// Transfermode/specific_MA_config/FB_Write_config_MA_06
/// This function block can be used to download the configuration of Motion App 6 ("ECO drive").
/// The specific parameters of this Motion App are the inputs of this FB and can be defined by the user. 
/// The function block uses the transfer mode to write this configuration to the Motion Terminal
/// and indicates the state of the download process.

FUNCTION_BLOCK FB_Write_config_MA_06
VAR_INPUT
	awBusDataFromVTEM 				: ARRAY [0..2] OF WORD;		(* 6 bytes of process data received from the Motion Terminal *)
END_VAR
	
VAR_IN_OUT
	awBusDataToVTEM 				: ARRAY [0..2] OF WORD; 	(* 6 bytes of process data sent to the Motion Terminal *)
END_VAR

VAR_INPUT
	xExecute 						: BOOL; 					(* has to be set to TRUE for a download and to FALSE to reset the function block after a download *)

	iParameterSet					: INT := 1; 				(* the parameter set to be written to, 1 by default *)
	
	// system parameters
		iInPortRetracted			: INT;						// Sensor port for detection of end position at pressurisation of outlet port 2 (retracted), value is number of the slot (beginning from 0 and including valve slots) * 10 + number of the port
		iInPortAdvanced				: INT;						// Sensor port for detection of end position at pressurisation of outlet port 4 (advanced), value is number of the slot (beginning from 0 and including valve slots) * 10 + number of the port

END_VAR

VAR_OUTPUT                  		
	iResponse 						: eTransferResponse; 		(* returns the status of the execution of the download process *)
	sCurrentValue 					: STRING; 					(* indicates which value of the array is currently treated (necessary to evaluate in case of error messages) *)
	xDownloadDone 					: BOOL; 					(* indicates whether the download was successful *)
	xDownloadError 					: BOOL := FALSE; 			(* indicates whether an error occurred during the transfer *)
END_VAR

VAR
	aTransferPackages				: ARRAY [0..100] OF stTransferPackage;
	fbdownloadMultipleParameters 	: FB_Download_Multiple_Parameters;
	iCurrentValue					: INT;
	fbWriteValueToWord 				: FB_Write_Value_To_Word;
END_VAR

(*****************************************************************************************************

Festo SE & Co. KG, Esslingen
Copyright (c) 2018. All rights reserved.

Product:            Motion Terminal VTEM
Description:        Function Block to download the parameters for Motion App 6 to the Motion Terminal

Object version:     2.00
Last change:        2019-03
======================================================================================================
                                       H I S T O R Y
======================================================================================================
Version:            2.00
Date:               2019-03
Change/Activity:    - created (#2368895)
Release:            3.5.7.230 (CODESYS 3.5.7.2, Lib version 3.0)
Author:             JEBU
======================================================================================================

*****************************************************************************************************)

// write the Motion App specific parameters into the struct
	//iInPortRetract
		aTransferPackages[0].iChannel := iParameterSet;
		aTransferPackages[0].iAddressedTarget := 6;
		aTransferPackages[0].iIndex := 70;
		aTransferPackages[0].iTransferValue := iInPortRetracted;
	
	//iInPortRetract
		aTransferPackages[1].iChannel := iParameterSet;
		aTransferPackages[1].iAddressedTarget := 6;
		aTransferPackages[1].iIndex := 71;
		aTransferPackages[1].iTransferValue := iInPortAdvanced;
	
	// define end of parameter list to be downloaded by setting all variables to 0 (end criterion for FB_Download_Multiple_Parameters)
		aTransferPackages[2].iChannel := 0;
		aTransferPackages[2].iAddressedTarget := 0;
		aTransferPackages[2].iIndex := 0;
		aTransferPackages[2].iTransferValue := 0;


// pre-check of the value for the parameter set
	IF xExecute = TRUE AND (iParameterSet < 1 OR iParameterSet > 5) THEN		// invalid input for the parameter set
		xDownloadDone := FALSE; 
		xDownloadError := TRUE; 
		iResponse := eTransferResponse.invalid_ParameterSet; 
		iCurrentValue := 0; 
		// send command 'stop'
		fbWriteValueToWord(iValue := 61, iStartBit := 0, iEndBit := 5, wDataWord := awBusDataToVTEM[0]); 			// ValveMode = 61
		fbWriteValueToWord(iValue := 0, iStartBit := 6, iEndBit := 15, wDataWord := awBusDataToVTEM[0]); 			// (empty)
		awBusDataToVTEM[1] := 0; 
		awBusDataToVTEM[2] := 0; 
		
	ELSE	
		// call the function block for multiple parameter download
			fbdownloadMultipleParameters(	xExecute := xExecute,
											awBusDataFromVTEM := awBusDataFromVTEM,
											aTransferPackages := aTransferPackages, 
											awBusDataToVTEM := awBusDataToVTEM,
											xDownloadDone => xDownloadDone,
											xDownloadError => xDownloadError,
											iResponse => iResponse,
											iCurrentValue => iCurrentValue);
	END_IF
	
	
// The current value output is needed if there is any invalid value in order to address it correctly.
// As the user doesn't work with indices in this function block, the current value is transformed to a string holding the name of the parameter.
	CASE iCurrentValue OF
		0: sCurrentValue := 'iInPortRetract';
		1: sCurrentValue := 'iInPortAdvanced';
		2: sCurrentValue := 'AllParametersWritten';
	END_CASE

END_FUNCTION_BLOCK

// Operation/FB_TeachInRun
/// This function block is designed to execute the teach-in run (Valve Mode 60) on a valve. 
/// Before executing the transfer mode, the Parameter 255 (Motion App to be tought in) is
/// parameterised with the value on the corresponding input.
/// After that the teach-in run is started and can be controlled via the input "iManualControl"
/// if the manual operation is possible for the selectes Motion App.

FUNCTION_BLOCK FB_TeachInRun
VAR_INPUT
	awBusDataFromVTEM				: ARRAY [0..2] OF WORD;				// 6 bytes of process data that is received from the Motion Terminal
END_VAR

VAR_IN_OUT
	awBusDataToVTEM					: ARRAY [0..2] OF WORD;				// 6 bytes of process data that is sent to the Motion Terminal
END_VAR

VAR_INPUT
	xEnable							: BOOL;								// has to be set to TRUE in order to operate the teach-in run on the valve, otherwise the teach-in run is stopped  
	iParameterSet					: INT;								// Parameter Set to be used for storing the learning data (0 = current parameter set, 1…5 = parameter set 1…5)
	iMotionAppToBeToughtIn			: INT;								// ID of the Motion App that is to be taught-in
	iOperatingMode					: INT;								// Sets operating mode of teach-in run (0 = Stop, 1 = Auto, 2 = Manual (only Motion App #11)
	iManualControl					: INT;								// Control input for manual execution of teach-in run (0 = Block, 1 = Advance, 2 = Retract, 3 = Exhaust)
	xAcknowledge					: BOOL;								// errors can be acknowledged (after they got inactive) with a rising edge at this input, while the FB is enabled
END_VAR

VAR_OUTPUT
	xDone							: BOOL;								// indicates that the teach-in run was finished successfully
	xError							: BOOL;								// indicates that an Error occured
	iResponse						: eResponseTeachInRun;				// returns the status of the TeachInRun function block
	sResponseDescription			: STRING;							// returns the status of the TeachInRun function block as string
	xWarning						: BOOL;								// indicates whether there is a warning returned by the teach-in run
	xRetractedEndPos_optional		: BOOL;								// only if digital sensors are installed (optional): indicates whether the retracted end position was reached (after outlet port 2 is pressurised)
	xAdvancedEndPos_optional		: BOOL;								// only if digital sensors are installed (optional): indicates whether the advanced end position was reached (after outlet port 4 is pressurised)
END_VAR

VAR
	// State machine variables
		iState						: INT := 10;						// Value for the local state machine
		xStateChange				: BOOL;								// TRUE if the state is to be changed
		iCommandNumber				: INT;								// Value for the command case

	// First Cycle variables
		iParameterSetFC				: INT;								// Variable to store value from first cycle
		iMotionAppToBeToughtInFC	: INT;								// Variable to store value from first cycle
		iOperatingModeFCC			: INT;								// Variable to store value from first cycle in state "Completed" or "Error"
		iManualControlFCC			: INT;								// Variable to store value from first cycle in state "Completed" or "Error"

	// Function block instances
		fbreadbitsfromword				: FB_Read_Bits_From_Word;			// 
		fbwritevaluetoword				: FB_Write_Value_To_Word;			//
		fbstateinterpreterteachinrun	: FB_StateInterpreter_TeachInRun;	//

	// Current Valve variables
		iCurrentValveMode			: INT;									// 
		iCurrentValveState			: INT;									//
		iCurrentAppState			: INT;									//
		iCurrentChannelTM			: INT;									//
		iCurrentAddressedTargetTM	: INT;									//
		iCurrentIndexTM				: INT;									//
		iCurrentValueTM				: INT;									//
		iCurrentTransferControlTM	: INT;									//
		
	// Misc variables
		xInputValid					: BOOL;									// TRUE if the values iParameterSet, iMotionAppToBeToughtIn and iOperatingMode are within valid range
		xInputConsistent			: BOOL;
		xInvalidCommand				: BOOL;
		iInvalidCommand				: INT;
		xNoValve					: BOOL;
		xWebConfigAccess			: BOOL;
		xInvalidMotionApp			: BOOL;
		
		xAcknowledgeLastCycle		: BOOL;
		
		xAcknowledgeCompleted		: BOOL;
		xReadyToComplete			: BOOL;									// Indicator which shows that no outdated response of the last executed learning trip is evaluated. 
		xStateFinished				: BOOL;
		xStateError					: BOOL;
		
		iReadParameterSet			: INT;
		iWriteParameterSet			: INT;
		xReturnReadParameterSet		: BOOL;
		
		iCounter					: INT;
		iCounterMax					: INT := 3000;
		
		xTeachInRunWasActive		: BOOL;
END_VAR

(*****************************************************************************************************

Festo SE & Co. KG, Esslingen
Copyright (c) 2019. All rights reserved.

Product:            Motion Terminal VTEM
Description:        Function block to execute the teach-in run

Object version:     1.05
Last change:        2020-12
======================================================================================================
                                       H I S T O R Y
======================================================================================================
Version:            1.05 
Date:               2020-12        
Change/Activity:    - integrated new app state return values #10 and #11 (#3800494)
Release:            3.5.7.236
Author:             JEBU
------------------------------------------------------------------------------------------------------
Version:            1.04 
Date:               2020-05        
Change/Activity:    - created (#2256363)
Release:            3.5.7.234
Author:             JEBU/MKLP
======================================================================================================

******************************************************************************************************)

// Read the current status of the the motion terminal
	fbreadbitsfromword(wData:= awBusDataFromVTEM[0], iStartBit:=0, iEndBit:= 5, iValue=> iCurrentValveMode, xError=> );						// read current valve mode
	fbreadbitsfromword(wData:= awBusDataFromVTEM[0], iStartBit:=6, iEndBit:= 7, iValue=> iCurrentValveState, xError=> );					// read current valve state

	IF iCurrentValveMode <> 63 THEN																										// Operating mode:
		fbreadbitsfromword(wData:= awBusDataFromVTEM[0], iStartBit:=8, iEndBit:= 15, iValue=> iCurrentAppState, xError=>);					// read app state
	ELSIF iCurrentValveMode = 63 THEN																									// Transfer mode:
		fbreadbitsfromword(wData:= awBusDataFromVTEM[0], iStartBit:= 8, iEndBit:= 12, iValue=> iCurrentChannelTM, xError=> );				// read current channel
		fbreadbitsfromword(wData:= awBusDataFromVTEM[0], iStartBit:= 13, iEndBit:= 15, iValue=> iCurrentTransferControlTM, xError=> );		// read current transfer control
		fbreadbitsfromword(wData:= awBusDataFromVTEM[1], iStartBit:= 0, iEndBit:= 7, iValue=> iCurrentAddressedTargetTM, xError=> );		// read current addressed target
		fbreadbitsfromword(wData:= awBusDataFromVTEM[1], iStartBit:= 8, iEndBit:= 15, iValue=> iCurrentIndexTM, xError=> );					// read current index
		fbreadbitsfromword(wData:= awBusDataFromVTEM[2], iStartBit:= 0, iEndBit:= 15, iValue=> iCurrentValueTM, xError=> );					// read current value
	END_IF
	
	IF iCurrentValveMode = 60 AND iState = 40 THEN
		fbstateinterpreterteachinrun.byActualAppState := INT_TO_BYTE(iCurrentAppState);
		
		fbstateinterpreterteachinrun();
				
		xRetractedEndPos_optional := fbstateinterpreterteachinrun.xRetractedEndPos_optional;
		xAdvancedEndPos_optional := fbstateinterpreterteachinrun.xAdvancedEndPos_optional;
		xWarning := fbstateinterpreterteachinrun.xWarning;
		iResponse := fbstateinterpreterteachinrun.iTeachInRunState;
	END_IF
//-----------------------------------------------------------------------------------------------------------

// Transition for RESETTING 
	IF xEnable = FALSE AND iState <> 10 AND iState <> 100 THEN
		xStateChange := TRUE;
		iState := 100;
	END_IF
//-----------------------------------------------------------------------------------------------------------

// Transition for WebConfig Access denied
	IF 	xWebConfigAccess = FALSE AND 
		xEnable = TRUE AND iState <> 10 AND 
		iCurrentValveMode = 61 AND iCurrentAppState = 10 THEN 	// The WebConfig has write permission -> access denied for the PLC
			xStateChange := TRUE;
			iState := 70;
			xWebConfigAccess := TRUE;
	END_IF
//-----------------------------------------------------------------------------------------------------------
	
// Check if input data is consisent (not in state 10 IDLE)
	IF 	xInputConsistent = TRUE  AND 
		xEnable = TRUE AND iState <> 10 AND iState <> 15 AND 
		(iParameterSet <> iParameterSetFC OR iMotionAppToBeToughtIn <> iMotionAppToBeToughtInFC OR (iState = 70 AND xStateChange = FALSE AND (iOperatingModeFCC <> iOperatingMode OR iManualControlFCC <> iManualControl))) THEN
			xStateChange := TRUE;
			iState := 70;		// Input data inconsistent
			xInputConsistent := FALSE;		
	END_IF
	
	IF xNoValve = FALSE AND 
	   xEnable = TRUE AND iState <> 10 AND iState <> 15 AND 
	   iCurrentValveMode = 61 AND iCurrentValveState = 1 AND iCurrentAppState = 15 THEN		// no Valve detected 
			xNoValve := TRUE;
			xStateChange := TRUE;
			iState := 70;
	END_IF
//-----------------------------------------------------------------------------------------------------------

// Local state machine
	CASE iState OF
		10:	// IDLE mode
			// code that is executed only in the first cycle of this state
				IF xStateChange = TRUE THEN
					xStateChange := FALSE;
				END_IF
			//-----------------------------------------------------------------------------------------------------------
			
			// code that is repeated every cycle in this state	
				iCommandNumber := 0;	// IDLE
				iResponse := eResponseTeachInRun.idle;
			//-----------------------------------------------------------------------------------------------------------
			
			// Transition
				IF xEnable = TRUE THEN
					xStateChange := TRUE;	// Leave this state
					iState := 15;
				END_IF
			//-----------------------------------------------------------------------------------------------------------

		15:	// check validity and save values of "first cycle"
			// code that is executed only in the first cycle of this state
				IF xStateChange = TRUE THEN
					xStateChange := FALSE;
					iResponse := eResponseTeachInRun.storing_first_cycle_input_data;
					xInputConsistent := TRUE;
					iParameterSetFC := iParameterSet;
					iMotionAppToBeToughtInFC := iMotionAppToBeToughtIn;
				END_IF
			//-----------------------------------------------------------------------------------------------------------
			
			// code that is repeated every cycle in this state	
				IF (iParameterSet >= 0 AND iParameterSet <= 5) AND (iMotionAppToBeToughtIn >= 1 AND iMotionAppToBeToughtIn <= 59) AND (iOperatingMode >= 0 AND iOperatingMode <= 3) THEN
					xInputValid := TRUE;
				ELSE
					xInputValid := FALSE;
				END_IF
			//-----------------------------------------------------------------------------------------------------------
			
			// Transition
				IF xInputValid = TRUE THEN
					xStateChange := TRUE;	// Leave this state
					iState := 20;
				ELSE
					xStateChange := TRUE;	// Leave this state
					iState := 70;			// Failure
				END_IF
			//-----------------------------------------------------------------------------------------------------------
		
		20:	// Resetting valve mode to 61
			// code that is executed only in the first cycle of this state
				IF xStateChange = TRUE THEN
					xStateChange := FALSE;
					iResponse := eResponseTeachInRun.resetting_valve_to_61;
				END_IF
			//-----------------------------------------------------------------------------------------------------------
			
			// code that is repeated every cycle in this state	
				IF iCurrentValveMode = 63 THEN
					iCommandNumber := 1;	// exit transfer mode
				ELSIF iCurrentValveMode <> 61 AND iCurrentValveMode <> 63 AND iCurrentValveState = eValveState.Running THEN
					iCommandNumber := 2;	// stop running motion apps
				END_IF 
			//-----------------------------------------------------------------------------------------------------------
			
			// Transition
				IF iCurrentValveMode = 61 AND iCurrentValveState = eValveState.configurable THEN
					xStateChange := TRUE;	// Leave this state
					iState := 30;
				ELSIF iCurrentValveState = eValveState.NotReady OR iCurrentValveState = eValveState.Failure THEN
					xStateChange := TRUE;
					iState := 70;
				END_IF
			//-----------------------------------------------------------------------------------------------------------

		30: // Sending command to read active ParameterSet
				// code that is executed only in the first cycle of this state
				IF xStateChange = TRUE THEN
					xStateChange := FALSE;
					xStateFinished := FALSE;
					iResponse := eResponseTeachInRun.ReadingActiveParameterSet;
					iCommandNumber := 3;	// read active ParameterSet
				END_IF
			//-----------------------------------------------------------------------------------------------------------
			
			// code that is repeated every cycle in this state
				IF iCurrentValveMode = 63 AND iCurrentChannelTM = 15 AND iCurrentAddressedTargetTM = 0 AND iCurrentIndexTM = 1 THEN
					xStateFinished := TRUE;
					iReadParameterSet := iCurrentValueTM;
				ELSE // timeout mechanism after <iCounterMax> cycles within this state
					iCounter := iCounter + 1;
					IF iCounter = iCounterMax THEN
						xStateError := TRUE;
					END_IF
				END_IF
				
				IF iParameterSet = 0 THEN
					iWriteParameterSet := iReadParameterSet;
				ELSE
					iWriteParameterSet := iParameterSet;
				END_IF
			//-----------------------------------------------------------------------------------------------------------
				
			// Transition
				IF xStateFinished = TRUE THEN
					xStateChange := TRUE;
					iState := 32;
				ELSIF xStateError = TRUE THEN
					xStateChange := TRUE;
					iState := 70;
				END_IF 					
			//-----------------------------------------------------------------------------------------------------------
			
		32: // Sending command to change active ParameterSet
				// code that is executed only in the first cycle of this state
				IF xStateChange = TRUE THEN
					xStateChange := FALSE;
					xStateFinished := FALSE;
					iResponse := eResponseTeachInRun.ChangingActiveParameterSet;
					iCommandNumber := 4;	// change ParameterSet
				END_IF
			//-----------------------------------------------------------------------------------------------------------
			
			// code that is repeated every cycle in this state
				IF iCurrentValveMode = 63 AND iCurrentChannelTM = 15 AND iCurrentAddressedTargetTM = 0 AND iCurrentIndexTM = 1 AND iCurrentValueTM = iWriteParameterSet THEN
					xStateFinished := TRUE;
				ELSIF iCurrentValveMode = 63 AND iCurrentTransferControlTM = 0 AND iCurrentChannelTM = 0 AND iCurrentAddressedTargetTM = 0 AND iCurrentIndexTM = 0 AND iCurrentValueTM = 5 THEN
					xStateError := TRUE;
				END_IF
			//-----------------------------------------------------------------------------------------------------------
				
			// Transition
				IF xStateFinished = TRUE THEN
					xStateChange := TRUE;
					iState := 34;
				ELSIF xStateError = TRUE THEN
					xStateChange := TRUE;
					iState := 70;
				END_IF 					
			//----------------------------------------------------------------------------------------------------------- 
			
		34:	// Sending command to write parameter 255 (motion app to be tought in)	
			// code that is executed only in the first cycle of this state
				IF xStateChange = TRUE THEN
					xStateChange := FALSE;
					xStateFinished := FALSE;
					iResponse := eResponseTeachInRun.writing_parameter_MotionAppToBeToughtIn;
					iCommandNumber := 5;	// write parameter 255
				END_IF
			//-----------------------------------------------------------------------------------------------------------
			
			// code that is repeated every cycle in this state
				IF iCurrentValveMode = 63 AND iCurrentChannelTM = iWriteParameterSet AND iCurrentAddressedTargetTM = 60 AND iCurrentIndexTM = 255 AND iCurrentValueTM = iMotionAppToBeToughtIn THEN
					xStateFinished := TRUE;
					iCommandNumber := 1; //Exit Transfermode
				ELSIF iCurrentValveMode = 63 AND iCurrentTransferControlTM = 0 AND iCurrentChannelTM = 0 AND iCurrentAddressedTargetTM = 0 AND iCurrentIndexTM = 0 AND iCurrentValueTM = 5 THEN
					xInvalidMotionApp := TRUE;
				END_IF
			//-----------------------------------------------------------------------------------------------------------
				
			// Transition
				IF iCurrentValveMode = 61 AND xStateFinished = TRUE THEN
					xStateChange := TRUE;
					iState := 40;
				ELSIF xInvalidMotionApp = TRUE THEN
					xStateChange := TRUE;
					iState := 70;
				END_IF 
			//-----------------------------------------------------------------------------------------------------------
			
		40:	// Running Teach-in run
			// code that is executed only in the first cycle of this state
				IF xStateChange = TRUE THEN
					xStateChange := FALSE;
					xStateFinished := FALSE;
					iResponse := eResponseTeachInRun.running_teachIn_run;
					xTeachInRunWasActive := TRUE;
				END_IF
			//-----------------------------------------------------------------------------------------------------------
			
			// code that is repeated every cycle in this state
				IF NOT (iResponse = eResponseTeachInRun.running_teachIn_run OR							// This query is neccessary because of the behaviour of the teach-in run, that 
						iResponse = eResponseTeachInRun.TeachInRun_partially_completed_only_2 OR		// at the start it responds the result of the last teach-in run that was executed.
						iResponse = eResponseTeachInRun.TeachInRun_partially_completed_only_4 OR		// Because of this the state would end immediately if the last executed teach-in run
						iResponse = eResponseTeachInRun.TeachInRun_completed OR							// was finished e. g. with "completed". So the Response has to become one of this
						iResponse = eResponseTeachInRun.TeachInRun_completed_with_limitations) THEN		// values to indicate that a new teach-in run was staretd.
					xReadyToComplete := TRUE;
				END_IF
			
				iCommandNumber := 6;			// run TeachInRun
				
				IF iCurrentValveMode = 61 AND iCurrentValveState = 1 AND iCurrentAppState <> 0 THEN		// invalid command was sent 
					IF iCurrentAppState = 16 THEN
						iResponse := eResponseTeachInRun.valve_self_calibration_running;
					ELSE
						xInvalidCommand := TRUE;
						iInvalidCommand := iCurrentAppState;
					END_IF
				END_IF
			//-----------------------------------------------------------------------------------------------------------
			
			// Transition
				IF (iResponse = eResponseTeachInRun.TeachInRun_completed OR iResponse = eResponseTeachInRun.TeachInRun_partially_completed_only_2 OR iResponse = eResponseTeachInRun.TeachInRun_partially_completed_only_4 OR iResponse = eResponseTeachInRun.TeachInRun_completed_with_limitations) 
					AND iCurrentValveMode = 60 AND xReadyToComplete = TRUE AND (iOperatingMode = 1 OR iOperatingMode = 2) THEN
					xStateChange := TRUE;
					iState := 60;
				ELSIF iCurrentValveState = eValveState.NotReady OR iCurrentValveState = eValveState.Failure OR xInvalidCommand = TRUE OR iResponse = eResponseTeachInRun.TeachInRun_error THEN
					xStateChange := TRUE;
					iState := 70;
				END_IF
			//-----------------------------------------------------------------------------------------------------------
			
		60: // completed
			// code that is executed only in the first cycle of this state
				IF xStateChange = TRUE THEN
					xStateChange := FALSE;
					xDone := TRUE;
					xError := FALSE;
					iOperatingModeFCC := iOperatingMode;
					iManualControlFCC := iManualControl;
					// Reseting Output comming from the Stateinterpreter (except xWaring)
					xRetractedEndPos_optional := FALSE;
					xAdvancedEndPos_optional := FALSE;
				END_IF
			//-----------------------------------------------------------------------------------------------------------
			
			// code that is repeated every cycle in this state
				iCommandNumber := 2;

			//-----------------------------------------------------------------------------------------------------------
			
			// Transition
				IF iOperatingModeFCC <> iOperatingMode OR iManualControlFCC <> iManualControl THEN
					xStateChange := TRUE;
					iState := 70;
					xInputConsistent := FALSE;
				END_IF
			//-----------------------------------------------------------------------------------------------------------
			
		70:	// error
			// code that is executed only in the first cycle of this state
				IF xStateChange = TRUE THEN
					xStateChange := FALSE;
					xStateError := FALSE;
					IF xTeachInRunWasActive = FALSE THEN
						iResponse := eResponseTeachInRun.error_occured_check_DiagnosticMemory;
					END_IF
					IF xDone = FALSE THEN
						iOperatingModeFCC := iOperatingMode;
						iManualControlFCC := iManualControl;
					END_IF;
					xDone := FALSE;
					xError := TRUE;
					// Reseting Output comming from the Stateinterpreter
					xRetractedEndPos_optional := FALSE;
					xAdvancedEndPos_optional := FALSE;
					xWarning := FALSE;
				END_IF
			//-----------------------------------------------------------------------------------------------------------
				
				// Choosing iCommandNumber
				IF iCurrentValveState = eValveState.NotReady AND ((xAcknowledge = TRUE AND xAcknowledgeLastCycle = FALSE) OR iCommandNumber = 8) THEN
					iCommandNumber := 8; 	// Send 62 on rising edge of xAcknowlegde
				ELSE
					IF iCurrentValveMode = 63 THEN
						iCommandNumber := 1;
					ELSE
						iCommandNumber := 2;
					END_IF
				END_IF
				xAcknowledgeLastCycle := xAcknowledge;
					
				// Error Output
				IF xWebConfigAccess = TRUE THEN
					iResponse :=  eResponseTeachInRun.access_denied_WebConfig;
					IF NOT (iCurrentValveMode = 61 AND iCurrentAppState = 10) THEN
						iResponse := eResponseTeachInRun.FB_needs_rising_edge_xEnable;
					END_IF
				
				ELSIF xNoValve = TRUE THEN
					iResponse := eResponseTeachInRun.no_valve_detected;	
					
				ELSIF iCurrentValveState = eValveState.Failure THEN 
					iResponse := eResponseTeachInRun.error_occured_check_DiagnosticMemory;	
				
				ELSIF (iCurrentValveState = eValveState.NotReady OR iCommandNumber = 8) AND xTeachInRunWasActive = FALSE THEN
					iResponse := eResponseTeachInRun.acknowledge_needed;
					xAcknowledgeCompleted := FALSE;
								
				ELSIF (iResponse = eResponseTeachInRun.acknowledge_needed OR xAcknowledgeCompleted = TRUE) AND iCurrentValveState = eValveState.Configurable THEN
					iResponse := eResponseTeachInRun.FB_needs_rising_edge_xEnable;
					xAcknowledgeCompleted := TRUE;
					
				ELSIF xInputConsistent = FALSE AND ((iParameterSet >= 0 AND iParameterSet <= 5) AND (iMotionAppToBeToughtIn >= 1 AND iMotionAppToBeToughtIn <= 59) AND (iOperatingMode >= 0 AND iOperatingMode <= 2) AND (iManualControl >= 0 AND iManualControl <= 3)) THEN
					iResponse := eResponseTeachInRun.FB_needs_rising_edge_xEnable;
								
				ELSIF xInvalidCommand = TRUE THEN
					iResponse := iInvalidCommand + 100;
					IF iResponse = eResponseTeachInRun.invalid_SetAppControl THEN
						xInvalidCommand := FALSE;
						xInputValid := FALSE;
					END_IF
					
				ELSIF xInputValid = FALSE THEN
					iResponse := eResponseTeachInRun.input_data_invalid;
					
				ELSIF xInvalidMotionApp = TRUE THEN
					iResponse := eResponseTeachInRun.Invalid_MotionAppToBeToughtIn;
				END_IF
				
			//-----------------------------------------------------------------------------------------------------------
			
			// Transition
				// Transition to Resetting above the Case-Statemachine
			//-----------------------------------------------------------------------------------------------------------
			
		100:// resetting - VTEM and Function Block
			// code that is executed only in the first cycle of this state
				IF xStateChange = TRUE THEN
					xStateChange := FALSE;
					iResponse := eResponseTeachInRun.resetting;
					
					IF iCurrentValveMode = 63 THEN
						iCommandNumber := 1;	// exit transfer mode
					ELSE
						iCommandNumber := 2;	// stop running motion apps
					END_IF
				END_IF
			//-----------------------------------------------------------------------------------------------------------
			
			// code that is repeated every cycle in this state	
				IF xReturnReadParameterSet = FALSE AND iCurrentValveMode = 61 AND iReadParameterSet <> 0 THEN
					iCommandNumber := 7; //write previous active parameterset
				END_IF
				
				IF xReturnReadParameterSet = FALSE AND iCurrentValveMode = 63 AND iCurrentChannelTM = 15 AND iCurrentAddressedTargetTM = 0 AND iCurrentIndexTM = 1 AND iCurrentValueTM = iReadParameterSet THEN
					xReturnReadParameterSet := TRUE;
				ELSIF xReturnReadParameterSet = FALSE AND iReadParameterSet = 0 THEN
					xReturnReadParameterSet := TRUE;
				END_IF

				IF xReturnReadParameterSet = TRUE THEN
					// resetting the valve to valve mode 61
					IF iCurrentValveMode = 63 THEN
						iCommandNumber := 1;	// exit transfer mode
					ELSE
						iCommandNumber := 2;	// stop running motion apps
					END_IF 
				END_IF
				
			//-----------------------------------------------------------------------------------------------------------
				
			// Transition
				IF iCommandNumber = 2 AND ((xReturnReadParameterSet = TRUE AND iCurrentValveMode = 61) OR iCurrentValveState = eValveState.NotReady OR iCurrentValveState = eValveState.Failure) THEN
					xStateChange := TRUE;
					iState := 10;	// IDLE
					
					// resetting the function block
					xInvalidCommand := FALSE;
					iReadParameterSet := 0;
					xReturnReadParameterSet := FALSE;
					xReadyToComplete := FALSE;
					xWebConfigAccess := FALSE;
					xNoValve := FALSE;
					xInvalidMotionApp := FALSE;
					xAcknowledgeCompleted := FALSE;
					xRetractedEndPos_optional := FALSE;
					xAdvancedEndPos_optional := FALSE;
					xWarning := FALSE;
					xDone := FALSE;
					xError := FALSE;
					xTeachInRunWasActive := FALSE;					
				END_IF
			//-----------------------------------------------------------------------------------------------------------
			
	END_CASE
//-----------------------------------------------------------------------------------------------------------

// Set output sResponse (corresponding to eResponseTeachInRun)

	CASE iResponse OF
		0: sResponseDescription := 'TeachInRun_reserved';
		1: sResponseDescription := 'TeachInRun_unlearned';
		2: sResponseDescription := 'TeachInRun_check_tubes';
		3: sResponseDescription := 'TeachInRun_choose_control';
		4: sResponseDescription := 'TeachInRun_tune_trajectory';
		5: sResponseDescription := 'TeachInRun_determine_reference_value';
		6: sResponseDescription := 'TeachInRun_identification';
		10: sResponseDescription := 'operable_with_reduced_performance';
		11: sResponseDescription := 'completed_with_limitations';
		12: sResponseDescription := 'TeachInRun_partially_completed_only_2';
		13: sResponseDescription := 'TeachInRun_partially_completed_only_4';
		14: sResponseDescription := 'TeachInRun_completed';
		15: sResponseDescription := 'TeachInRun_error';
		101: sResponseDescription := 'invalid_SetValveMode';
		102: sResponseDescription := 'invalid_SetAppControl';
		103: sResponseDescription := 'invalid_SetAppOption';
		104: sResponseDescription := 'invalid_SetPointValue1';
		105: sResponseDescription := 'invalid_SetPointValue2';
		106: sResponseDescription := 'invalid_configuration';
		110: sResponseDescription := 'access_denied_WebConfig';
		111: sResponseDescription := 'access_denied_saving_parameterisation';
		112: sResponseDescription := 'no_license_for_this_MA';
		113: sResponseDescription := 'all_licenses_in_use';
		114: sResponseDescription := 'invalid_license_file';
		115: sResponseDescription := 'no_valve_detected';
		116: sResponseDescription := 'valve_self_calibration_running';
		210: sResponseDescription := 'idle';
		215: sResponseDescription := 'storing_first_cycle_input_data';
		220: sResponseDescription := 'resetting_valve_to_61';
		230: sResponseDescription := 'ReadingActiveParameterSet';
		232: sResponseDescription := 'ChangingActiveParameterSet';
		234: sResponseDescription := 'writing_parameter_MotionAppToBeToughtIn';
		240: sResponseDescription := 'running_teachIn_run';
		270: sResponseDescription := 'error_occured_check_DiagnosticMemory';
		271: sResponseDescription := 'input_data_invalid';
		272: sResponseDescription := 'FB_needs_rising_edge_xEnable';
		273: sResponseDescription := 'acknowledge_needed';
		274: sResponseDescription := 'Invalid_MotionAppToBeToughtIn';
		300: sResponseDescription := 'resetting';
	END_CASE
//-----------------------------------------------------------------------------------------------------------

// Command section
	CASE iCommandNumber OF
		0:	// IDLE
			;
			
		1:	// 	exit transfer mode
			fbwritevaluetoword(iValue:=63, iStartBit:=0, iEndBit:=5, wDataWord:=awBusDataToVTEM[0], xError=> );							// Valve Mode = 63
			fbwritevaluetoword(iValue:=0, iStartBit:=6, iEndBit:=7, wDataWord:=awBusDataToVTEM[0], xError=> );							// 0 (unused)
			fbwritevaluetoword(iValue:=0, iStartBit:=8, iEndBit:=12, wDataWord:=awBusDataToVTEM[0], xError=> );							// Channel = 0 (ignored)
			fbwritevaluetoword(iValue:=3, iStartBit:=13, iEndBit:=15, wDataWord:=awBusDataToVTEM[0], xError=> );						// Transfer Control = Exit transfer mode (3)
			fbwritevaluetoword(iValue:=0, iStartBit:=0, iEndBit:=7, wDataWord:=awBusDataToVTEM[1], xError=> );							// Addressed Target = 0 (ignored)
			fbwritevaluetoword(iValue:=0, iStartBit:=8, iEndBit:=15, wDataWord:=awBusDataToVTEM[1], xError=> );							// Index = 0 (ignored)
			fbwritevaluetoword(iValue:=0, iStartBit:=0, iEndBit:=15, wDataWord:=awBusDataToVTEM[2], xError=> );							// Value = 0 (ignored)
			
		2:	// stop running motion apps
			fbwritevaluetoword(iValue:=61, iStartBit:=0, iEndBit:=5, wDataWord:=awBusDataToVTEM[0], xError=> );							// Valve Mode = 61 (stop)
			fbwritevaluetoword(iValue:=0, iStartBit:=6, iEndBit:=7, wDataWord:=awBusDataToVTEM[0], xError=> );							// App Control = 0 (unused)
			fbwritevaluetoword(iValue:=0, iStartBit:=8, iEndBit:=15, wDataWord:=awBusDataToVTEM[0], xError=> );							// App Option = 0 (unused)
			fbwritevaluetoword(iValue:=0, iStartBit:=0, iEndBit:=15, wDataWord:=awBusDataToVTEM[1], xError=> );							// Setpoint Value 1 = 0 (unused)
			fbwritevaluetoword(iValue:=0, iStartBit:=0, iEndBit:=15, wDataWord:=awBusDataToVTEM[2], xError=> );							// Setpoint Value 2 = 0 (unused)
			
		3:	//	read active parameterSet
			fbwritevaluetoword(iValue:=63, iStartBit:=0, iEndBit:=5, wDataWord:=awBusDataToVTEM[0], xError=> );							// Valve Mode = 63
			fbwritevaluetoword(iValue:=15, iStartBit:=8, iEndBit:=12, wDataWord:=awBusDataToVTEM[0], xError=> );						// Channel = 15
			fbwritevaluetoword(iValue:=2, iStartBit:=13, iEndBit:=15, wDataWord:=awBusDataToVTEM[0], xError=> );						// Transfer Control = Upload (2)
			fbwritevaluetoword(iValue:=0, iStartBit:=0, iEndBit:=7, wDataWord:=awBusDataToVTEM[1], xError=> );							// Addressed Target = 0
			fbwritevaluetoword(iValue:=1, iStartBit:=8, iEndBit:=15, wDataWord:=awBusDataToVTEM[1], xError=> );							// Index = 1 

		4:	//	change active parameterSet
			fbwritevaluetoword(iValue:=63, iStartBit:=0, iEndBit:=5, wDataWord:=awBusDataToVTEM[0], xError=> );							// Valve Mode = 63
			fbwritevaluetoword(iValue:=15, iStartBit:=8, iEndBit:=12, wDataWord:=awBusDataToVTEM[0], xError=> );						// Channel = 15
			fbwritevaluetoword(iValue:=1, iStartBit:=13, iEndBit:=15, wDataWord:=awBusDataToVTEM[0], xError=> );						// Transfer Control = Download (1)
			fbwritevaluetoword(iValue:=0, iStartBit:=0, iEndBit:=7, wDataWord:=awBusDataToVTEM[1], xError=> );							// Addressed Target = 0
			fbwritevaluetoword(iValue:=1, iStartBit:=8, iEndBit:=15, wDataWord:=awBusDataToVTEM[1], xError=> );							// Index = 1 
			fbwritevaluetoword(iValue:=iWriteParameterSet, iStartBit:=0, iEndBit:=15, wDataWord:=awBusDataToVTEM[2], xError=> );		// Value = iParameterSet
			
		5:	//	write value from input iMotionAppToBeToughtIn to Parameter 255
			fbwritevaluetoword(iValue:=63, iStartBit:=0, iEndBit:=5, wDataWord:=awBusDataToVTEM[0], xError=> );							// Valve Mode = 63
			fbwritevaluetoword(iValue:=iWriteParameterSet, iStartBit:=8, iEndBit:=12, wDataWord:=awBusDataToVTEM[0], xError=> );		// Channel = iParameterSet
			fbwritevaluetoword(iValue:=1, iStartBit:=13, iEndBit:=15, wDataWord:=awBusDataToVTEM[0], xError=> );						// Transfer Control = Download (1)
			fbwritevaluetoword(iValue:=60, iStartBit:=0, iEndBit:=7, wDataWord:=awBusDataToVTEM[1], xError=> );							// Addressed Target = Teach-in run (60)
			fbwritevaluetoword(iValue:=255, iStartBit:=8, iEndBit:=15, wDataWord:=awBusDataToVTEM[1], xError=> );						// Index = 255 (Motion App to be tought in)
			fbwritevaluetoword(iValue:=iMotionAppToBeToughtIn, iStartBit:=0, iEndBit:=15, wDataWord:=awBusDataToVTEM[2], xError=> );	// Value = iMotionAppToBeToughtIn

		6:	// running the teach-in run
			fbWriteValueToWord(iValue := 60, iStartBit := 0, iEndBit := 5, wDataWord := awBusDataToVTEM[0]); 							// iSetValveMode = 60
			fbWriteValueToWord(iValue := iOperatingMode, iStartBit := 6, iEndBit := 7, wDataWord := awBusDataToVTEM[0]); 				// bySetAppControl = iOperatingMode
			fbWriteValueToWord(iValue := 0, iStartBit := 8, iEndBit := 15, wDataWord := awBusDataToVTEM[0]); 							// bySetAppOption = 0
		
			awBusDataToVTEM[1] := INT_TO_WORD(iManualControl);																			// SetpointValue1 = iManualControl
			awBusDataToVTEM[2] := 0;

		7:	// change active parameterSet back to previous value
			fbwritevaluetoword(iValue:=63, iStartBit:=0, iEndBit:=5, wDataWord:=awBusDataToVTEM[0], xError=> );							// Valve Mode = 63
			fbwritevaluetoword(iValue:=15, iStartBit:=8, iEndBit:=12, wDataWord:=awBusDataToVTEM[0], xError=> );						// Channel = 15
			fbwritevaluetoword(iValue:=1, iStartBit:=13, iEndBit:=15, wDataWord:=awBusDataToVTEM[0], xError=> );						// Transfer Control = Download (1)
			fbwritevaluetoword(iValue:=0, iStartBit:=0, iEndBit:=7, wDataWord:=awBusDataToVTEM[1], xError=> );							// Addressed Target = 0
			fbwritevaluetoword(iValue:=1, iStartBit:=8, iEndBit:=15, wDataWord:=awBusDataToVTEM[1], xError=> );							// Index = 1 
			fbwritevaluetoword(iValue:=iReadParameterSet, iStartBit:=0, iEndBit:=15, wDataWord:=awBusDataToVTEM[2], xError=> );			// Value = iParameterSet
		
		8:	// Send 62 (Acknowledge)
			fbWriteValueToWord(iValue := 62, iStartBit := 0, iEndBit := 5, wDataWord := awBusDataToVTEM[0]); 							// ValveMode = 62
			fbWriteValueToWord(iValue := 0, iStartBit := 6, iEndBit := 15, wDataWord := awBusDataToVTEM[0]); 							// (empty)
			awBusDataToVTEM[1] := 0; 																									// (empty)
			awBusDataToVTEM[2] := 0;																									// (empty)
	END_CASE
//-----------------------------------------------------------------------------------------------------------

END_FUNCTION_BLOCK

// StateInterpreter/FB_StateInterpreter_TeachInRun
/// The variable "byActualAppState" is an output of the FB_ValveControl that is used differently in each Motion App.
/// This function block interprets the "AppState" output of the FB_ValveControl if the Tech-In Run (Valve Mode 60) is running.
/// The valve mode specific values are derived from the "byActualAppState".

FUNCTION_BLOCK FB_StateInterpreter_TeachInRun
VAR_INPUT
	byActualAppState 			: BYTE; 					// output of the FB_ValveControl
END_VAR
VAR_OUTPUT
	xRetractedEndPos_optional	: BOOL;  					// only if digital sensors are installed (optional): indicates whether the retracted end position was reached (after outlet port 2 is pressurised)
	xAdvancedEndPos_optional	: BOOL;  					// only if digital sensors are installed (optional): indicates whether the advanced end position was reached (after outlet port 4 is pressurised)
	iTeachInRunState			: eResponseTeachInRun;		// indicates the state of the Teach-In run as a numeric value
	sTeachInRunState			: STRING;					// indicates the state of the Teach-In run as a text
	xWarning					: BOOL; 					// indicates whether there is a warning returned by the Teach-In run
END_VAR
VAR
	fbReadBitsFromByte			: FB_Read_Bits_From_Byte;
	byRetractedEndPos			: BYTE;
	byAdvancedEndPos			: BYTE;
	byTeachInState		 		: BYTE;  					
	byWarning					: BYTE;
END_VAR

(*****************************************************************************************************

Festo SE & Co. KG, Esslingen
Copyright (c) 2018. All rights reserved.

Product:            Motion Terminal VTEM
Description:        Function block for interpreting the app state of the Teach-In Run 

Object version:     1.03
Last change:        2020-12
======================================================================================================
                                       H I S T O R Y
======================================================================================================
Version:            1.03
Date:               2020-12
Change/Activity:    - added new values 10 and 11 (#3800494)
Release:            3.5.7.236
Author:             JEBU
------------------------------------------------------------------------------------------------------
Version:            1.02
Date:               2020-03
Change/Activity:    - created
Release:            3.5.7.234
Author:             JEBU/MKLP
======================================================================================================

*****************************************************************************************************)

// read the Motion App specific values from the ActualAppState byte
fbReadBitsFromByte(byData := byActualAppState, iStartBit := 0, iEndBit := 0, byValue => byRetractedEndPos);
xRetractedEndPos_optional :=  BYTE_TO_BIT(byRetractedEndPos);

fbReadBitsFromByte(byData := byActualAppState, iStartBit := 2, iEndBit := 2, byValue => byAdvancedEndPos); 
xAdvancedEndPos_optional :=  BYTE_TO_BIT(byAdvancedEndPos);

fbReadBitsFromByte(byData := byActualAppState, iStartBit := 3, iEndBit := 6, byValue => byTeachInState);
iTeachInRunState := byTeachInState;

fbReadBitsFromByte(byData := byActualAppState, iStartBit := 7, iEndBit := 7, byValue => byWarning);
xWarning := BYTE_TO_BIT(byWarning);

CASE iTeachInRunState OF
	0:	sTeachInRunState := 'reserved';
	1:	sTeachInRunState := 'unlearned';
	2:	sTeachInRunState := 'check_tubes';
	3:	sTeachInRunState := 'choose_control';
	4:	sTeachInRunState := 'tune_trajectory';
	5:	sTeachInRunState := 'determine_reference_value';
	6:	sTeachInRunState := 'identification';
	10: sTeachInRunState := 'operable_with_reduced_performance';
	11: sTeachInRunState := 'completed_with_limitations';
	12:	sTeachInRunState := 'partially_completed_only_2';
	13:	sTeachInRunState := 'partially_completed_only_4';
	14:	sTeachInRunState := 'completed';
	15:	sTeachInRunState := 'error';
END_CASE

END_FUNCTION_BLOCK

// Transfermode/specific_MA_config/FB_Write_config_MA_33
/// This function block can be used to download the configuration of Motion App 33 ("Positioning").
/// The specific parameters of this Motion App are the inputs of this FB and can be defined by the user. 
/// The function block uses the transfer mode to write this configuration to the Motion Terminal
/// and indicates the state of the download process.

FUNCTION_BLOCK FB_Write_config_MA_33
VAR_INPUT
	awBusDataFromVTEM 				: ARRAY [0..2] OF WORD;				// 6 bytes of process data received from the Motion Terminal
END_VAR

VAR_IN_OUT
	awBusDataToVTEM 				: ARRAY [0..2] OF WORD; 			// 6 bytes of process data sent to the Motion Terminal	
END_VAR

VAR_INPUT
	xExecute 											: BOOL; 		// has to be set to TRUE for a download and to FALSE to reset the function block after a download

	iParameterSet										: INT := 1; 	// the parameter set to be written to, 1 by default
	
	// system parameters
		iTubingLengthAt2 								: INT; 			// length of the tubing connected to outlet port 2 of the valve [1 digit = 1 mm]
	 	iTubingLengthAt4 								: INT;			// length of the tubing connected to outlet port 4 of the valve [1 digit = 1 mm]
	 	iTubingInnerDiameterAt2							: INT;  		// inner diameter of the tubing connected to outlet port 2 of the valve [1 digit = 0.01 mm]
	 	iTubingInnerDiameterAt4							: INT;			// inner diameter of the tubing connected to outlet port 4 of the valve [1 digit = 0.01 mm]
	 	iDriveType 										: INT;			// type of the drive/cylinder/... that is to be operated by the valve ->  see list of drive types at support portal (www.festo.com/sp/)
	 	iDriveStroke 									: INT; 			// stroke of the drive/cylinder/... that is to be operated by the valve [1 digit = 1 mm for linear drives, 1 digit = 1° for rotary drives]
		iInstallationPositionDrive 						: INT;  	 	// inclination of the cylinder with reference to a horizontal installation position [1 digit = 0.01°, positive values = advancing upwards]
		iOffsetAxisZeroPoint							: INT;			// offset of the mechanical stop "retracted" to the retracted end of the nominal stroke [1 digit = 1 mm]
		iInPortFullStrokeMeas							: INT;			// sensor port for positioning measurement over the entire working stroke; value is number of the slot (beginning from 0 and including valve slots) * 10 + number of the port, -1 for usage of partial stroke measurement   
		iInPortPartStrokeMeasRet						: INT;			// sensor port for position measurement over the part of the working stroke at the retracted end; value is number of the slot (beginning from 0 and including valve slots) * 10 + number of the port, -1 if no sensor is connected
		iInPortPartStrokeMeasAdv						: INT;			// sensor port for position measurement over the part of the working stroke at the advanced end; value is number of the slot (beginning from 0 and including valve slots) * 10 + number of the port, -1 if no sensor is connected
	
	// application parameters                               	
		iLoad			 								: INT;			// mass that is to be moved by the drive (retracting and advancing) [1 digit = 0.01 kg]
		iDampingTimeForTargetPositionReached			: INT;			// condition for feedback "Target position reached": actual position remains within the tolerance range around the target position for the specified time [1 digit = 0.01 s]
		iDurationOfThresholdExceedanceForError			: INT;			// condition for following error: Threshold value is exceeded for longer than the configured duration [1 digit = 0.001 s]
		iToleranceForTargetPositionReached				: INT;			// condition for feedback "Target Position Reached": permissible deviation of the actual position from the target position [1 digit = 0.1 mm]
		iMaxVelocityGeneral			 					: INT;			// maximum permissible velocity, independent of the direction of movement (general limitation; further limiting by setpoint value) [1 digit = 0.01 m/s]
		iMaxAcceleration								: INT;			// maximum permissible acceleration in direction of movement [1 digit = 0.1 m/s²]
		iMaxDeceleration								: INT;			// maximum permissible acceleration against the direction of movement [1 digit = 0.1 m/s²]
		iMaxJerk										: INT;			// maximum permissible jerk in direction of movement [1 digit = 0.1 m/s³]
		iOffsetProjectZeroPoint							: INT;			// offset to the reference point for target and actual positions to the axis zero point [1 digit = 1 mm]
		iOffsetSoftLimitNegEndRet						: INT;			// offset to lower "stop" of the desired working stroke to the axis zero point [1 digit = 1 mm]
		iOffsetSoftLimitPosEndAdv						: INT;			// offset to upper "stop" of the desired working stroke to the axis zero point  [1 digit = 1 mm]

		iDistTargPosWithConstVeloRet					: INT;			// Contact case: Distance to target position in retracting direction, on which the configured final velocity is to be applied
		iFinalVeloContactCaseRet						: INT;			// Contact case: Final velocity at contact in retracting direction
		iDistTargPosWithConstVeloAdv					: INT;			// Contact case: Distance to target position in advancing direction, on which the configured final velocity is to be applied
		iFinalVeloContactCaseAdv						: INT;			// Contact case: Final velocity at contact in advancing direction

		iMeanPressureLevel								: INT;			// mean pressure level [1 digit = 0.1 bar rel.]
		iThreshPosFollowError							: INT; 			// condition for following error: Actual position deviates from the planned trajectory by more than the threshold value for at least the configured duration [1 digit = 1 mm]  
		iTreshVeloFollowError							: INT; 			// condition for following error: Actual velocity deviates from the planned trajectory by more than the threshold value for at least the configured duration [1 digit = 0.001 m/s]
		iSoftStartFunction								: INT;			// Pre-pressurisation of cylinder chambers; 0 = disabled, 1 = enabled
		iEndPositionMonitoring							: INT;			// 0 = active for both end positions, 1 = active for retracted end position, 2 = active for advanced end position, 3 = inactive 
		xOptionPressureBuildUpIntoMechEndPos			: BOOL;			// 0 = Setpoint values are only accepted within the actual effective stroke, 1 = Allow setpoint values outside the actual effective stroke in order to build up pressure into the mechanical end position

	// tuning parameters
		iOptControllerGainRelative						: INT;			// Optional tuning parameter for controller gain (relative adjustment of the internally used value) [1 digit = 1%]
		iOptDampingOfSystemAbsolute						: INT;			// Optional tuning parameter for damping of the controlled system (absolute adjustment of the internally used value [1 digit = 0.01]
		iOptPliabilityRelative							: INT;			// Optional tuning parameter for pliability (relative adjustment of the internally used value) [1 digit = 1%]
		iOptReductionOfPilotControlRelative				: INT;			// Optional tuning parameter for reduction of pilot control (relative adjustment of the internally used value) [1 digit = 1%]
		iOptCoulombFritionInAccountRelative				: INT;			// Optional tuning parameter for coulomb friction taken into account(relative adjustment of the internally used value) [1 digit = 1%]

END_VAR
VAR_OUTPUT
	iResponse 											: eTransferResponse;	// returns the status of the execution of the download process *)
	sCurrentValue 										: STRING; 		// indicates which value of the array is currently treated (necessary to evaluate in case of error messages) *)
	xDownloadDone 										: BOOL; 		// indicates whether the download was successful *)
	xDownloadError 										: BOOL := FALSE;	// indicates whether an error occurred during the transfer *)
END_VAR

VAR
	aTransferPackages									: ARRAY [0..100] OF stTransferPackage;
	fbdownloadMultipleParameters 						: FB_Download_Multiple_Parameters;
	iCurrentValue										: INT;
	fbWriteValueToWord 									: FB_Write_Value_To_Word;
END_VAR

(*****************************************************************************************************

Festo SE & Co. KG, Esslingen
Copyright (c) 2021. All rights reserved.

Product:            Motion Terminal VTEM
Description:        Function block to download the parameters for Motion App 33 to the Motion Terminal

Object version:     1.02
Last change:        2021-03
======================================================================================================
Version:            1.02
Date:               2021-03
Change/Activity:    - included new application parameters (#4102819)
Release:            3.5.7.236 (CODESYS 3.5.7.2, Lib version 3.6)
Author:             JEBU
------------------------------------------------------------------------------------------------------
Version:            1.01
Date:               2020-09
Change/Activity:    - created (#2256322)
Release:            3.5.7.235 (CODESYS 3.5.7.2, Lib version 3.5)
Author:             JEBU
======================================================================================================

*****************************************************************************************************)

// write the Motion App specific parameters into the struct
	//iTubingLengthAt2
		aTransferPackages[0].iChannel := iParameterSet;
		aTransferPackages[0].iAddressedTarget := 33;
		aTransferPackages[0].iIndex := 12;
		aTransferPackages[0].iTransferValue := iTubingLengthAt2;
		
	//iTubingLengthAt4
		aTransferPackages[1].iChannel := iParameterSet;
		aTransferPackages[1].iAddressedTarget := 33;
		aTransferPackages[1].iIndex := 13;
		aTransferPackages[1].iTransferValue := iTubingLengthAt4;
		
	//iTubingInnerDiameterAt2
		aTransferPackages[2].iChannel := iParameterSet;
		aTransferPackages[2].iAddressedTarget := 33;
		aTransferPackages[2].iIndex := 14;
		aTransferPackages[2].iTransferValue := iTubingInnerDiameterAt2;
		
	//iTubingInnerDiameterAt4
		aTransferPackages[3].iChannel := iParameterSet;
		aTransferPackages[3].iAddressedTarget := 33;
		aTransferPackages[3].iIndex := 15;
		aTransferPackages[3].iTransferValue := iTubingInnerDiameterAt4;
		
	//iDriveType
		aTransferPackages[4].iChannel := iParameterSet;
		aTransferPackages[4].iAddressedTarget := 33;
		aTransferPackages[4].iIndex := 20;
		aTransferPackages[4].iTransferValue := iDriveType;
		
	//iDriveStroke
		aTransferPackages[5].iChannel := iParameterSet;
		aTransferPackages[5].iAddressedTarget := 33;
		aTransferPackages[5].iIndex := 21;
		aTransferPackages[5].iTransferValue := iDriveStroke;
		
	//iInstallationPositionDrive
		aTransferPackages[6].iChannel := iParameterSet;
		aTransferPackages[6].iAddressedTarget := 33;
		aTransferPackages[6].iIndex := 60;
		aTransferPackages[6].iTransferValue := iInstallationPositionDrive;
		
	//iOffsetAxisZeroPoint
		aTransferPackages[7].iChannel := iParameterSet;
		aTransferPackages[7].iAddressedTarget := 33;
		aTransferPackages[7].iIndex := 61;
		aTransferPackages[7].iTransferValue := iOffsetAxisZeroPoint;
		
	//iInPortFullStrokeMeas		
		aTransferPackages[8].iChannel := iParameterSet;
		aTransferPackages[8].iAddressedTarget := 33;
		aTransferPackages[8].iIndex := 80;
		aTransferPackages[8].iTransferValue := iInPortFullStrokeMeas;
		
	//iInPortPartStrokeMeasRet	
		aTransferPackages[9].iChannel := iParameterSet;
		aTransferPackages[9].iAddressedTarget := 33;
		aTransferPackages[9].iIndex := 75;
		aTransferPackages[9].iTransferValue := iInPortPartStrokeMeasRet;
		
	//iInPortPartStrokeMeasAdv	
		aTransferPackages[10].iChannel := iParameterSet;
		aTransferPackages[10].iAddressedTarget := 33;
		aTransferPackages[10].iIndex := 76;
		aTransferPackages[10].iTransferValue := iInPortPartStrokeMeasAdv;
		
	//iLoad
		aTransferPackages[11].iChannel := iParameterSet;
		aTransferPackages[11].iAddressedTarget := 33;
		aTransferPackages[11].iIndex := 100;
		aTransferPackages[11].iTransferValue := iLoad;
		
	//iDampingTimeForTargetPositionReached
		aTransferPackages[12].iChannel := iParameterSet;
		aTransferPackages[12].iAddressedTarget := 33;
		aTransferPackages[12].iIndex := 124;
		aTransferPackages[12].iTransferValue := iDampingTimeForTargetPositionReached;
		
	//iDurationOfThresholdExceedanceForError
		aTransferPackages[13].iChannel := iParameterSet;
		aTransferPackages[13].iAddressedTarget := 33;
		aTransferPackages[13].iIndex := 126;
		aTransferPackages[13].iTransferValue := iDurationOfThresholdExceedanceForError;
		
	//iToleranceForTargetPositionReached	
		aTransferPackages[14].iChannel := iParameterSet;
		aTransferPackages[14].iAddressedTarget := 33;
		aTransferPackages[14].iIndex := 141;
		aTransferPackages[14].iTransferValue := iToleranceForTargetPositionReached;
		
	// iMaxVelocityGeneral
		aTransferPackages[15].iChannel := iParameterSet;
		aTransferPackages[15].iAddressedTarget := 33;
		aTransferPackages[15].iIndex := 142;
		aTransferPackages[15].iTransferValue := iMaxVelocityGeneral;
		
	//iMaxAcceleration
		aTransferPackages[16].iChannel := iParameterSet;
		aTransferPackages[16].iAddressedTarget := 33;
		aTransferPackages[16].iIndex := 144;
		aTransferPackages[16].iTransferValue := iMaxAcceleration;
		
	//iMaxDecelaration
		aTransferPackages[17].iChannel := iParameterSet;
		aTransferPackages[17].iAddressedTarget := 33;
		aTransferPackages[17].iIndex := 146;
		aTransferPackages[17].iTransferValue := iMaxDeceleration;
		
	//iMaxJerk
		aTransferPackages[18].iChannel := iParameterSet;
		aTransferPackages[18].iAddressedTarget := 33;
		aTransferPackages[18].iIndex := 148;
		aTransferPackages[18].iTransferValue := iMaxJerk;
		
	//iOffsetProjectZeroPoint
		aTransferPackages[19].iChannel := iParameterSet;
		aTransferPackages[19].iAddressedTarget := 33;
		aTransferPackages[19].iIndex := 150;
		aTransferPackages[19].iTransferValue := iOffsetProjectZeroPoint;
		
	//iOffsetSoftLimitNegEndRet
		aTransferPackages[20].iChannel := iParameterSet;
		aTransferPackages[20].iAddressedTarget := 33;
		aTransferPackages[20].iIndex := 151;
		aTransferPackages[20].iTransferValue := iOffsetSoftLimitNegEndRet;
		
	//iOffsetSoftLimitPosEndAdv
		aTransferPackages[21].iChannel := iParameterSet;
		aTransferPackages[21].iAddressedTarget := 33;
		aTransferPackages[21].iIndex := 152;
		aTransferPackages[21].iTransferValue := iOffsetSoftLimitPosEndAdv;
		
	//iDistTargPosWithConstVeloRet
		aTransferPackages[22].iChannel := iParameterSet;
		aTransferPackages[22].iAddressedTarget := 33;
		aTransferPackages[22].iIndex := 153;
		aTransferPackages[22].iTransferValue := iDistTargPosWithConstVeloRet;
		
	//iFinalVeloContactCaseRet
		aTransferPackages[23].iChannel := iParameterSet;
		aTransferPackages[23].iAddressedTarget := 33;
		aTransferPackages[23].iIndex := 155;
		aTransferPackages[23].iTransferValue := iFinalVeloContactCaseRet;
		
	//iDistTargPosWithConstVeloAdv
		aTransferPackages[24].iChannel := iParameterSet;
		aTransferPackages[24].iAddressedTarget := 33;
		aTransferPackages[24].iIndex := 154;
		aTransferPackages[24].iTransferValue := iDistTargPosWithConstVeloAdv;
		
	//iFinalVeloContactCaseAdv
		aTransferPackages[25].iChannel := iParameterSet;
		aTransferPackages[25].iAddressedTarget := 33;
		aTransferPackages[25].iIndex := 156;
		aTransferPackages[25].iTransferValue := iFinalVeloContactCaseAdv;

	//iMeanPressureLevel
		aTransferPackages[26].iChannel := iParameterSet;
		aTransferPackages[26].iAddressedTarget := 33;
		aTransferPackages[26].iIndex := 184;
		aTransferPackages[26].iTransferValue := iMeanPressureLevel;
		
	// iThreshPosFollowError
		aTransferPackages[27].iChannel := iParameterSet;
		aTransferPackages[27].iAddressedTarget := 33;
		aTransferPackages[27].iIndex := 204;
		aTransferPackages[27].iTransferValue := iThreshPosFollowError;
		
	// iTreshVeloFollowError
		aTransferPackages[28].iChannel := iParameterSet;
		aTransferPackages[28].iAddressedTarget := 33;
		aTransferPackages[28].iIndex := 205;
		aTransferPackages[28].iTransferValue := iTreshVeloFollowError;
		
	// iSoftStartFunction
		aTransferPackages[29].iChannel := iParameterSet;
		aTransferPackages[29].iAddressedTarget := 33;
		aTransferPackages[29].iIndex := 222;
		aTransferPackages[29].iTransferValue := iSoftStartFunction;
		
	// iEndPositionMonitoring
		aTransferPackages[30].iChannel := iParameterSet;
		aTransferPackages[30].iAddressedTarget := 33;
		aTransferPackages[30].iIndex := 224;
		aTransferPackages[30].iTransferValue := iEndPositionMonitoring;
		
	// xOptionPressureBuildUpIntoMechEndPos
		aTransferPackages[31].iChannel := iParameterSet;
		aTransferPackages[31].iAddressedTarget := 33;
		aTransferPackages[31].iIndex := 225;
		aTransferPackages[31].iTransferValue := BOOL_TO_INT(xOptionPressureBuildUpIntoMechEndPos);

	// iOptControllerGainRelative
		aTransferPackages[32].iChannel := iParameterSet;
		aTransferPackages[32].iAddressedTarget := 33;
		aTransferPackages[32].iIndex := 230;
		aTransferPackages[32].iTransferValue := iOptControllerGainRelative;
			
	// iOptDampingOfSystemAbsolute				
		aTransferPackages[33].iChannel := iParameterSet;
		aTransferPackages[33].iAddressedTarget := 33;
		aTransferPackages[33].iIndex := 231;
		aTransferPackages[33].iTransferValue := iOptDampingOfSystemAbsolute;
			
	// iOptPliabilityRelative						
		aTransferPackages[34].iChannel := iParameterSet;
		aTransferPackages[34].iAddressedTarget := 33;
		aTransferPackages[34].iIndex := 232;
		aTransferPackages[34].iTransferValue := iOptPliabilityRelative;
			
	// iOptReductionOfPilotControlRelative		
		aTransferPackages[35].iChannel := iParameterSet;
		aTransferPackages[35].iAddressedTarget := 33;
		aTransferPackages[35].iIndex := 233;
		aTransferPackages[35].iTransferValue := iOptReductionOfPilotControlRelative;
			
	// iOptCoulombFritionInAccountRelative		
		aTransferPackages[36].iChannel := iParameterSet;
		aTransferPackages[36].iAddressedTarget := 33;
		aTransferPackages[36].iIndex := 234;
		aTransferPackages[36].iTransferValue := iOptCoulombFritionInAccountRelative;

	// define end of parameter list to be downloaded by setting all variables to 0 (end criterion for FB_Download_Multiple_Parameters)
		aTransferPackages[37].iChannel := 0;
		aTransferPackages[37].iAddressedTarget := 0;
		aTransferPackages[37].iIndex := 0;
		aTransferPackages[37].iTransferValue := 0;


// pre-check of the value for the parameter set
IF xExecute = TRUE AND (iParameterSet < 1 OR iParameterSet > 5) THEN		// invalid input for the parameter set
	xDownloadDone := FALSE; 
	xDownloadError := TRUE; 
	iResponse := eTransferResponse.invalid_ParameterSet; 
	iCurrentValue := 0; 
	// send command 'stop'
	fbWriteValueToWord(iValue := 61, iStartBit := 0, iEndBit := 5, wDataWord := awBusDataToVTEM[0]); 			// ValveMode = 61
	fbWriteValueToWord(iValue := 0, iStartBit := 6, iEndBit := 15, wDataWord := awBusDataToVTEM[0]); 			// (empty)
	awBusDataToVTEM[1] := 0; 
	awBusDataToVTEM[2] := 0; 
	
ELSE	
	// call the function block for multiple parameter download
	fbdownloadMultipleParameters(	xExecute := xExecute,
									awBusDataFromVTEM := awBusDataFromVTEM,
									awBusDataToVTEM := awBusDataToVTEM,
									aTransferPackages := aTransferPackages,  
									xDownloadDone => xDownloadDone,
									xDownloadError => xDownloadError,
									iResponse => iResponse,
									iCurrentValue => iCurrentValue); 
END_IF
	
	
// The current value output is needed if there is any invalid value in order to address it correctly.
// As the user doesn't work with indices in this function block, the current value is transformed to a string holding the name of the parameter.
CASE iCurrentValue OF
	0: sCurrentValue := 'iTubingLengthAt2';
	1: sCurrentValue := 'iTubingLengthAt4';
	2: sCurrentValue := 'iTubingInnerDiameterAt2';
	3: sCurrentValue := 'iTubingInnerDiameterAt4';
	4: sCurrentValue := 'iDriveType';
	5: sCurrentValue := 'iDriveStroke';
	6: sCurrentValue := 'iInstallationPositionDrive';
	7: sCurrentValue := 'iOffsetAxisZeroPoint';
	8: sCurrentValue := 'iInPortFullStrokeMeas';
	9: sCurrentValue := 'iInPortPartStrokeMeasRet';
	10: sCurrentValue := 'iInPortPartStrokeMeasAdv';
	11: sCurrentValue := 'iLoad';
	12: sCurrentValue := 'iDampingTimeForTargetPositionReached';
	13: sCurrentValue := 'iDurationOfThresholdExceedanceForError';
	14: sCurrentValue := 'iToleranceForTargetPositionReached';
	15: sCurrentValue := 'iMaxVelocityGeneral';
	16: sCurrentValue := 'iMaxAcceleration';
	17: sCurrentValue := 'iMaxDeceleration';
	18: sCurrentValue := 'iMaxJerk';
	19: sCurrentValue := 'iOffsetProjectZeroPoint';
	20: sCurrentValue := 'iOffsetSoftLimitNegEndRet';
	21: sCurrentValue := 'iOffsetSoftLimitPosEndAdv';
	22: sCurrentValue := 'iDistTargPosWithConstVeloRet';
	23: sCurrentValue := 'iFinalVeloContactCaseRet';
	24: sCurrentValue := 'iDistTargPosWithConstVeloAdv';
	25: sCurrentValue := 'iFinalVeloContactCaseAdv';
	26: sCurrentValue := 'iMeanPressureLevel';
	27: sCurrentValue := 'iThreshPosFollowError';
	28: sCurrentValue := 'iTreshVeloFollowError';
	29: sCurrentValue := 'iSoftStartFunction';
	30: sCurrentValue := 'iEndPositionMonitoring';
	31: sCurrentValue := 'xOptionPressureBuildUpIntoMechEndPos';
	32: sCurrentValue := 'iOptControllerGainRelative';			
	33: sCurrentValue := 'iOptDampingOfSystemAbsolute';			
	34: sCurrentValue := 'iOptPliabilityRelative';					
	35: sCurrentValue := 'iOptReductionOfPilotControlRelative';	
	36: sCurrentValue := 'iOptCoulombFritionInAccountRelative';	
	37: sCurrentValue := 'AllParametersWritten';
END_CASE

END_FUNCTION_BLOCK

// Transfermode/FB_Download_Single_Parameter
/// This function block can be used to run the transfer mode of the Motion Terminal in order to download a single value.
/// The value to be downloaded needs to be addressed, indicating the channel, the addressed target and the index of the value.

FUNCTION_BLOCK FB_Download_Single_Parameter
VAR_INPUT
	awBusDataFromVTEM 		: ARRAY [0..2] OF WORD; 		(* 6 bytes of process data received from the Motion Terminal *)
END_VAR	

VAR_IN_OUT
	awBusDataToVTEM 		: ARRAY [0..2] OF WORD; 		(* 6 bytes of process data sent to the Motion Terminal *)
END_VAR

VAR_INPUT	
	xExecute 				: BOOL;							(* has to be set to TRUE for a download and to FALSE to reset the function block after a download *)
	                                                                
	iChannel 				: INT;							(* the channel the value is to be written to (see documentation for details) *)
	iAddressedTarget 		: INT; 							(* the target by which the parameter value is to be used (was "iAddressedApp" in former versions) (see documentation for details) *)
	iIndex 					: INT;							(* the index of the parameter (see documentation for details) *)
	iDownloadValue 			: INT;  						(* the value to be downloaded *)
END_VAR

VAR_OUTPUT
	iResponse 				: eTransferResponse;			(* returns the status of the execution of the download process *)
	xDownloadDone 			: BOOL := FALSE; 				(* indicates whether the download was successful *)
	xDownloadError 			: BOOL := FALSE; 				(* indicates whether an error occurred during the transfer *)
END_VAR

VAR
	iRecValveMode 			: INT;
	iRecValveStatus 		: eValveState;
	
	iCommandNumber			: INT; 							(* indicates the command to be executed *)

	fbWriteValueToWord		: FB_Write_Value_To_Word;
	fbReadBitsFromWord 		: FB_Read_Bits_From_Word;
	iRecChannel				: INT;
	iRecTransferCtrl		: INT;
	iRecAddressedTargetType	: INT;
	iRecIndex				: INT;
	iRecDownloadValue		: INT;
	
	iAppStatus				: INT;
	iLastChannel			: INT;
	iLastAddressedTarget	: INT;
	iLastIndex				: INT;
	iLastTransferValue		: INT;
	xFirstCycle				: BOOL := TRUE;					(* avoids the analysis of the data from the Motion Terminal in the first cycle as they are not a reaction to the current command *)
	xTransferComplete		: BOOL;
	xSavingSuccessful 		: BOOL;
	iFCChannel				: INT;							(* value at the channel input while first cycle of the fb *)
	iFCAddressedTarget		: INT;							(* value at the addressed app input while first cycle of the fb *)
	iFCIndex				: INT;							(* value at the index input while first cycle of the fb *) 
	iFCDownloadValue		: INT;							(* value at the download value input while first cycle of the fb*)
	xFCSavePersistent		: BOOL;
	xInputConsistent		: BOOL;							(* stays TRUE if the input values do not change until the download job is done *)
	xInputValid				: BOOL;							(* TRUE if the input values are within the correct range for each input *)
END_VAR

(*****************************************************************************************************

Festo SE & Co. KG, Esslingen
Copyright (c) 2018. All rights reserved.

Product:            Motion Terminal VTEM
Description:        Function block to download a single parameter to the Motion Terminal

Object version:     2.01
Last change:        2019-07
======================================================================================================
                                       H I S T O R Y
======================================================================================================
Version:            2.01
Date:               2019-07        
Change/Activity:    - adjusted range for iChannel from 255 to 31 (#2510540)
					- adapted functionality for transfer mode on slots without valves (#2957509)
					- added new enum value (#3104444)
Release:            3.5.7.234 (CODESYS 3.5.7.2, Lib version 3.4)
Author:             MKLP/JEBU
------------------------------------------------------------------------------------------------------
Version:            2.00
Date:               2019-03
Change/Activity:    - changed awBusDataToVTEM into VAR_IN_OUT (#2368965)
                    - fixed bug that caused "exit transfer mode" even if xExecute is FALSE (#2181575)
                    - added value 7 to list of invalid commands (#2318899)
Release:            3.5.7.230 (CODESYS 3.5.7.2, Lib version 3.0)
Author:             JEBU/MKLP
------------------------------------------------------------------------------------------------------
Version:            1.01
Date:               2018-11
Change/Activity:    - adjusted value range of iChannel and iAddressedTarget to 0...255 (#2181575)
Release:            3.5.7.221 (CODESYS 3.5.7.2, Lib version 2.1)
Author:             JEBU
------------------------------------------------------------------------------------------------------
Version:            1.00
Date:               2017
Change/Activity:    - created
Release:            3.5.7.22 (CODESYS 3.5.7.2, Lib version 2.0)
Author:             HLBG
======================================================================================================

*****************************************************************************************************)

// read the ValveMode and the ValveState of the Motion Terminal
fbReadBitsFromWord(wData := awBusDataFromVTEM[0], iStartBit := 0, iEndBit := 5, iValue => iRecValveMode);
fbReadBitsFromWord(wData := awBusDataFromVTEM[0], iStartBit := 6, iEndBit := 7, iValue => iRecValveStatus);

// A rising edge at xExecute indicates that new values are to be written, xExecute must be TRUE during the whole download procedure
IF xExecute = TRUE THEN
	
	// pre-analysis of the input data before caring about the transfer
	IF xFirstCycle = TRUE THEN
		// store the command that was given in the first cycle
		iFCChannel := iChannel;
		iFCAddressedTarget := iAddressedTarget;
		iFCIndex := iIndex;
		iFCDownloadValue := iDownloadValue;
		
		IF iChannel < 0 OR iChannel > 31 THEN
			iResponse := eTransferResponse.invalid_Channel;
			xInputValid := FALSE;
		ELSIF iAddressedTarget < 0 OR iAddressedTarget > 255 THEN
 			iResponse := eTransferResponse.invalid_AddressedTarget;
			xInputValid := FALSE;
		ELSIF iIndex < 0 OR iIndex > 255 THEN
 			iResponse := eTransferResponse.invalid_Index;
			xInputValid := FALSE;
		ELSE
			xInputValid := TRUE;
			xInputConsistent := TRUE;
		END_IF
		
	ELSE	// xFirstCycle = FALSE
		// check whether the current command is still the same compared to the command at the rising edge of xExecute
		IF iFCChannel = iChannel AND iFCAddressedTarget = iAddressedTarget AND iFCIndex = iIndex AND iFCDownloadValue = iDownloadValue THEN
			xInputConsistent := TRUE;
 		ELSE
			xInputConsistent := FALSE;
			iResponse := eTransferResponse.FB_needs_rising_edge_xExecute;
		END_IF
	END_IF

	IF xInputConsistent = TRUE AND xInputValid = TRUE THEN
		IF iRecValveStatus = eValveState.Running THEN		// a Motion App is running
			iResponse := eTransferResponse.preparing_transfer;
			iCommandNumber := 3; 					// command 'stop'
			xDownloadError := FALSE;
			
		ELSE	// The transfer mode can be used as the ValveStatus is not RUNNING
			IF iRecValveMode <> 63 AND xDownloadDone = FALSE THEN	// The transfer mode is currently not active and the value is not downloaded yet
				// check whether the WebConfig blocks the access to transfer mode
				fbReadBitsFromWord(wData := awBusDataFromVTEM[0], iStartBit := 8, iEndBit := 15, iValue => iAppStatus);
				IF iRecValveMode = 61 AND iAppStatus = 10 THEN 	// access denied by WebConfig
					xDownloadError := TRUE;
					iResponse := eTransferResponse.access_denied_WebConfig;
					iCommandNumber := 3; 			// do nothing (here: command 'stop')
				ELSIF iRecValveMode = 61 AND iAppStatus = 11 THEN 	// access denied due to an active saving process
					xDownloadError := TRUE; 
					iResponse := eTransferResponse.access_denied_saving; 
					iCommandNumber := 3; 			// do nothing (here: command 'stop')
				ELSIF iRecValveMode = 61 AND iAppStatus = 15 THEN 	// no valve detected
					xDownloadError := TRUE; 
					iResponse := eTransferResponse.no_valve_detected; 
					iCommandNumber := 1; 			// keep downloading (here: command 'download') In a Firmware older than 4.16(E) an empty valve keep sending ValveMode 61 and AppStatus 15. In Firmware 4.16(E) the message changes with a tranfer
				ELSIF iRecValveMode = 61 AND iAppStatus = 0 AND xTransferComplete = TRUE THEN 
					// The value is downloaded and the transfer mode has been closed properly
					xDownloadDone := TRUE;
					xDownloadError := FALSE;
					iCommandNumber := 3; 			// command 'stop' to remain the valve stopped
				ELSE	// ready to start transfer mode
					xDownloadError := FALSE;
					iResponse := eTransferResponse.transferring;
					iCommandNumber := 1; 			// command 'download' for the value
				END_IF
		
			ELSIF iRecValveMode = 63 AND xDownloadDone = FALSE THEN	// The transfer mode is active, but the value is not downloaded yet
				fbReadBitsFromWord(wData := awBusDataFromVTEM[0], iStartBit := 8, iEndBit := 12, iValue => iRecChannel);
				fbReadBitsFromWord(wData := awBusDataFromVTEM[0], iStartBit := 13, iEndBit := 15, iValue => iRecTransferCtrl);
				fbReadBitsFromWord(wData := awBusDataFromVTEM[1], iStartBit := 0, iEndBit := 7, iValue => iRecAddressedTargetType);
				fbReadBitsFromWord(wData := awBusDataFromVTEM[1], iStartBit := 8, iEndBit := 15, iValue => iRecIndex);
				iRecDownloadValue := WORD_TO_INT(awBusDataFromVTEM[2]);
		 
				IF iChannel = iRecChannel AND iRecTransferCtrl = 1 AND iRecAddressedTargetType = iAddressedTarget AND iRecIndex = iIndex AND  iDownloadValue = iRecDownloadValue THEN
				// The download command for the parameter was mirrored by the Motion Terminal, the download has been confirmed
					xTransferComplete := TRUE;	// ready for the saving process
					xDownloadError := FALSE;
					// notice the last downloaded parameter
					iLastChannel := iChannel;
					iLastAddressedTarget := iAddressedTarget;
					iLastIndex := iIndex;
					iLastTransferValue := iDownloadValue;
			 
					iCommandNumber := 2; 			// exit transfer mode
					iResponse := eTransferResponse.transfer_successful;
				
				ELSIF iRecChannel = 0 AND iRecTransferCtrl = 0 AND iRecAddressedTargetType = 0 AND iRecIndex = 0 AND iRecDownloadValue <> 0 AND xFirstCycle = FALSE THEN
					// An invalid command was sent when using the transfer mode
					
					iCommandNumber := 1; 			// command 'download' for the value
					xDownloadError := TRUE;
					
					CASE iRecDownloadValue OF	// indicates the type of the invalid command
						1: 	iResponse := eTransferResponse.invalid_Channel; 
						2: 	iResponse := eTransferResponse.invalid_TransferControl;	// this should never happen 
						3: 	iResponse := eTransferResponse.invalid_AddressedTarget;
						4: 	iResponse := eTransferResponse.invalid_Index; 
						5: 	iResponse := eTransferResponse.invalid_TransferValue;
						6: 	iResponse := eTransferResponse.invalid_combination;
						7:	iResponse := eTransferResponse.access_denied_DataInUse;
						8:	iResponse := eTransferResponse.no_data_empty_slot;
					END_CASE

				ELSE	// A different value is treated in transfer mode or the command was mirrored wrong
					iCommandNumber := 1; 		// command 'download' for the value
					xDownloadError := FALSE;
					iResponse := eTransferResponse.transferring;
				END_IF
			
			ELSE // xDownloadDone = TRUE
				IF iLastChannel = iChannel AND iLastAddressedTarget = iAddressedTarget AND iLastIndex = iIndex AND iLastTransferValue = iDownloadValue THEN
					// The FB is still active although the value is already downloaded
					iResponse := eTransferResponse.transfer_successful;
					xDownloadError := FALSE;
					iCommandNumber := 3; 		// do nothing (here: command 'stop', MAs remain stopped)
				ELSE
					// Another value was inserted to the FB without resetting the internal state with a falling edge at xExecute before
					iResponse := eTransferResponse.FB_needs_rising_edge_xExecute;
					xDownloadError := TRUE;
					iCommandNumber := 2; 		// do nothing (here: command 'exit transfer mode')
				END_IF
			END_IF
		END_IF
		
	ELSE // xInputValid = FALSE OR xInputConsistent = FALSE
		xDownloadDone := FALSE;
		xDownloadError := TRUE;
		IF iRecValveMode = 63 THEN
			iCommandNumber := 2; 				// command 'exit transfer mode'
		ELSE
			iCommandNumber := 3;				// command 'stop'
		END_IF

	END_IF
	xFirstCycle := FALSE; 
	
ELSIF xExecute = FALSE AND xFirstCycle = FALSE THEN	// falling edge at input xExecute, reseting the function block
	IF iRecValveMode = 63 THEN
		iCommandNumber := 2;						// exit transfer mode
	ELSE
		xFirstCycle := TRUE;
		xDownloadDone := FALSE;
		xDownloadError := FALSE;
		xTransferComplete := FALSE;
		iResponse := eTransferResponse.ready_for_new_transfer;
		iCommandNumber := 0;						// do nothing (idle)
	END_IF

ELSIF xExecute = FALSE AND xFirstCycle = TRUE THEN	// idle mode for the function block
	iResponse := eTransferResponse.ready_for_new_transfer;
	iCommandNumber := 0;	
END_IF

CASE iCommandNumber OF
	0: // idle

	1: // download the value that is addressed and specified in the input of this FB
		fbWriteValueToWord(iValue := 63, iStartBit := 0, iEndBit := 5, wDataWord := awBusDataToVTEM[0]); 											// ValveMode = 63
		fbWriteValueToWord(iValue := 0, iStartBit := 6, iEndBit := 7, wDataWord := awBusDataToVTEM[0]); 											// (empty)
		fbWriteValueToWord(iValue := iChannel, iStartBit := 8, iEndBit := 12, wDataWord := awBusDataToVTEM[0]); 									// Channel
		fbWriteValueToWord(iValue := 1, iStartBit := 13, iEndBit := 15, wDataWord := awBusDataToVTEM[0]); 											// TransferControl = download
		fbWriteValueToWord(iValue := iAddressedTarget, iStartBit := 0, iEndBit := 7, wDataWord := awBusDataToVTEM[1]);								// AddressedTarget
		fbWriteValueToWord(iValue := iIndex, iStartBit := 8, iEndBit := 15, wDataWord := awBusDataToVTEM[1]); 										// Index
		
		awBusDataToVTEM[2] := INT_TO_WORD(iDownloadValue);
	
	2: // exit transfer mode
		fbWriteValueToWord(iValue := 63, iStartBit := 0, iEndBit := 5, wDataWord := awBusDataToVTEM[0]); 											// ValveMode = 63
		fbWriteValueToWord(iValue := 0, iStartBit := 6, iEndBit := 7, wDataWord := awBusDataToVTEM[0]); 											// (empty)
		fbWriteValueToWord(iValue := iChannel, iStartBit := 8, iEndBit := 12, wDataWord := awBusDataToVTEM[0]); 									// Channel
		fbWriteValueToWord(iValue := 3, iStartBit := 13, iEndBit := 15, wDataWord := awBusDataToVTEM[0]); 											// TransferControl = exit

		awBusDataToVTEM[1] := 0;
		awBusDataToVTEM[2] := 0;

	3: // stop all Motion Apps
		fbWriteValueToWord(iValue := 61, iStartBit := 0, iEndBit := 5, wDataWord := awBusDataToVTEM[0]); 											// ValveMode = 61
		fbWriteValueToWord(iValue := 0, iStartBit := 6, iEndBit := 15, wDataWord := awBusDataToVTEM[0]); 											// (empty)

		awBusDataToVTEM[1] := 0;
		awBusDataToVTEM[2] := 0;
END_CASE

END_FUNCTION_BLOCK

// Transfermode/FB_Upload_Multiple_Parameters
/// This function block can be used to run the transfer mode of the Motion Terminal in order to upload multiple values.

FUNCTION_BLOCK FB_Upload_Multiple_Parameters
VAR_INPUT
	awBusDataFromVTEM 		: ARRAY [0..2] OF WORD; 		(* 6 bytes of process data received from the Motion Terminal *)
END_VAR

VAR_IN_OUT
	awBusDataToVTEM 		: ARRAY [0..2] OF WORD; 		(* 6 bytes of process data sent to the Motion Terminal *)
END_VAR
	
VAR_INPUT	
	xExecute 				: BOOL;							(* has to be set to TRUE for an upload and to FALSE to reset the function block after an upload *)
END_VAR

VAR_OUTPUT
	iResponse 				: eTransferResponse;			(* returns the status of the execution of the upload process *)
	iCurrentValue 			: INT; 							(* indicates which array index is currently treated (necessary to evaluate in case of error messages) *)
	xUploadDone 			: BOOL; 						(* indicates whether the upload was successful *)
	xUploadError 			: BOOL; 						(* indicates whether an error occurred during the transfer *)
END_VAR

VAR_IN_OUT
	aTransferPackages 		: ARRAY[0..100] OF stTransferPackage;
END_VAR

VAR
	iRecValveMode 			: INT;
	iRecValveStatus 		: eValveState;
	iCommandNumber			: INT; 							(* indicates the command to be executed *)

	fbWriteValueToWord		: FB_Write_Value_To_Word;
	fbReadBitsFromWord 		: FB_Read_Bits_From_Word;
	iRecChannel				: INT;
	iRecTransferCtrl		: INT;
	iRecAddressedTargetType	: INT;
	iRecIndex				: INT;
	iRecTransferValue		: INT;
	iAppStatus				: INT;
	xFirstCycle				: BOOL := TRUE;
	xTransferComplete		: BOOL;
	aFCTransferPackages		: ARRAY [0..100] OF stTransferPackage;
	iLength					: INT;
	iFCLength				: INT;
	xInputValid				: BOOL;
	xInputConsistent		: BOOL;
	i						: INT;
	xStopPending			: BOOL;							// if TRUE the function block waits for the response from the motion terminal, that the transfer mode was quit
END_VAR

(*****************************************************************************************************

Festo SE & Co. KG, Esslingen
Copyright (c) 2018. All rights reserved.

Product:            Motion Terminal VTEM
Description:        Function block to upload multiple parameters from the Motion Terminal

Object version:     2.01
Last change:        2019-07
======================================================================================================
                                       H I S T O R Y
======================================================================================================
Version:            2.01
Date:               2019-07        
Change/Activity:    - adjusted range for iChannel from 255 to 31 (#2510540)
					- validity check shows first wrong element and stops the procedure (#2526112)
					- reintegrated sourcecode (#2521433)
					- adapted functionality for transfer mode on slots without valves (#2957509)
					- added new enum value (#3104444)
Release:            3.5.7.234 (CODESYS 3.5.7.2, Lib version 3.4)
Author:             MKLP/JEBU
------------------------------------------------------------------------------------------------------
Version:            2.00
Date:               2019-03
Change/Activity:    - changed awBusDataToVTEM into VAR_IN_OUT (#2368965)
                    - fixed bug that caused "exit transfer mode" even if xExecute is FALSE (#2181575)
                    - added value 7 to list of invalid commands (#2318899)
Release:            3.5.7.230 (CODESYS 3.5.7.2, Lib version 3.0)
Author:             JEBU/MKLP
------------------------------------------------------------------------------------------------------
Version:            1.02
Date:               2018-12
Change/Activity:    - fixed a bug regarding the stability of the function block (#2258021)
Release:            3.5.7.222 (CODESYS 3.5.7.2, Lib version 2.2)
Author:             JEBU
------------------------------------------------------------------------------------------------------
Version:            1.01
Date:               2018-11
Change/Activity:    - adjusted value range of iChannel and iAddressedTarget to 0...255 (#2181575)
Release:            3.5.7.221 (CODESYS 3.5.7.2, Lib version 2.1)
Author:             JEBU
------------------------------------------------------------------------------------------------------
Version:            1.00
Date:               2017
Change/Activity:    - created
Release:            3.5.7.22 (CODESYS 3.5.7.2, Lib version 2.0)
Author:             HLBG
=======================================================================================================

******************************************************************************************************)

// read the ValveMode and the ValveState of the Motion Terminal
fbReadBitsFromWord(wData := awBusDataFromVTEM[0], iStartBit := 0, iEndBit := 5, iValue => iRecValveMode);
fbReadBitsFromWord(wData := awBusDataFromVTEM[0], iStartBit := 6, iEndBit := 7, iValue => iRecValveStatus);

// A rising edge at xExecute indicates that new values are to be read, xExecute must be TRUE during the whole upload procedure
IF xExecute = TRUE THEN
	
	// pre-analysis of the input data before caring about the transfer
	IF xFirstCycle = TRUE THEN
		// reset StopPending	
		xStopPending := FALSE;
		
		// store the parameter array that was given in the first cycle
		aFCTransferPackages := aTransferPackages;
		
		// get the length of the parameter array
		iLength := 0;
		WHILE (aTransferPackages[iLength].iChannel <> 0 OR aTransferPackages[iLength].iAddressedTarget <> 0 OR aTransferPackages[iLength].iIndex <> 0 OR aTransferPackages[iLength].iTransferValue <> 0) DO
			iLength := iLength + 1;
		END_WHILE
		iFCLength := iLength;
				
		// check the single data items of the array
		xInputValid := TRUE;
		xInputConsistent := TRUE;
		
		FOR i := 0 TO iLength DO
			IF aTransferPackages[i].iChannel < 0 OR aTransferPackages[i].iChannel > 31 THEN
				iResponse := eTransferResponse.invalid_Channel;
				iCurrentValue := i;
				xInputValid := FALSE;
				EXIT;
			ELSIF aTransferPackages[i].iAddressedTarget < 0 OR aTransferPackages[i].iAddressedTarget > 255 THEN
				iResponse := eTransferResponse.invalid_AddressedTarget;
				iCurrentValue := i;
				xInputValid := FALSE;
				EXIT;
			ELSIF aTransferPackages[i].iIndex < 0 OR aTransferPackages[i].iIndex > 255 THEN
				iResponse := eTransferResponse.invalid_Index;
				iCurrentValue := i;
				xInputValid := FALSE;
				EXIT;
			END_IF
		END_FOR
		
	ELSE	// xFirstCycle = FALSE
		// check whether the current command is still the same compared to the command at the rising edge of xExecute
		
		// get the length of the parameter array
		iLength := 0;
		WHILE (aTransferPackages[iLength].iChannel <> 0 OR aTransferPackages[iLength].iAddressedTarget <> 0 OR aTransferPackages[iLength].iIndex <> 0 OR aTransferPackages[iLength].iTransferValue <> 0) DO
			iLength := iLength + 1;
		END_WHILE
		
		// check length and content of the array by comparing it to the array of the first cycle
		IF iFCLength <> iLength THEN
			xInputConsistent := FALSE;
			iResponse := eTransferResponse.FB_needs_rising_edge_xExecute;
  		ELSE
			FOR i := 0 TO iLength DO
				IF aFCTransferPackages[i].iChannel <> aTransferPackages[i].iChannel THEN
					xInputConsistent := FALSE;
					iResponse := eTransferResponse.FB_needs_rising_edge_xExecute;
				ELSIF aFCTransferPackages[i].iAddressedTarget <> aTransferPackages[i].iAddressedTarget THEN
					xInputConsistent := FALSE;
					iResponse := eTransferResponse.FB_needs_rising_edge_xExecute;
				ELSIF aFCTransferPackages[i].iIndex <> aTransferPackages[i].iIndex THEN
					xInputConsistent := FALSE;
					iResponse := eTransferResponse.FB_needs_rising_edge_xExecute;
				END_IF
			END_FOR
		END_IF
	END_IF 		// end of pre-analysis of the input data

	IF xInputConsistent = TRUE AND xInputValid = TRUE THEN
		IF iRecValveStatus = eValveState.Running THEN		// a Motion App is running
			iResponse := eTransferResponse.preparing_transfer;
			iCommandNumber := 3; 					// command 'stop'
			xUploadError := FALSE;
			
		ELSE	// The transfer mode can be used as the ValveStatus is not RUNNING
			IF iCommandNumber = 1 THEN // If transfer started with a virtual valve, eNum will be overwritten
				iResponse := eTransferResponse.transferring;
			END_IF
			
			IF iRecValveMode <> 63 AND xUploadDone = FALSE THEN	// The transfer mode is currently not active and the values are not uploaded yet
				// check whether the WebConfig blocks the access to transfer mode
				fbReadBitsFromWord(wData := awBusDataFromVTEM[0], iStartBit := 8, iEndBit := 15, iValue => iAppStatus);
				IF iRecValveMode = 61 AND iAppStatus = 10 THEN 		// access denied by WebConfig
					iResponse := eTransferResponse.access_denied_WebConfig; 
					xUploadError := TRUE;
					iCommandNumber := 3; 			// do nothing (here: command 'stop')
				ELSIF iRecValveMode = 61 AND iAppStatus = 11 THEN 	// access denied due to an active saving process
					xUploadError := TRUE;
					iResponse := eTransferResponse.access_denied_saving;
					iCommandNumber := 3; 			// do nothing (here: command 'stop')
				ELSIF iRecValveMode = 61 AND iAppStatus = 15 THEN 	// no valve detected
					xUploadError := TRUE;
					iResponse := eTransferResponse.no_valve_detected; 
					iCommandNumber := 1; 			// keep uploading (here: command 'upload') In a Firmware older than 4.16(E) an empty valve keep sending ValveMode 61 and AppStatus 15. In Firmware 4.16(E) the message changes with a tranfer
				ELSIF iRecValveMode = 61 AND iAppStatus = 0 AND xTransferComplete = TRUE THEN
					// All values are uploaded and the transfer mode has been closed properly
					xUploadDone := TRUE;
					xUploadError := FALSE;
					iCommandNumber := 3; 			// command 'stop' to remain the valve stopped
				ELSE	// ready to start transfer mode
					iResponse := eTransferResponse.transferring;
					xUploadError := FALSE;
					iCommandNumber := 1; 			// command 'upload' for the current value
				END_IF
		
			ELSIF iRecValveMode = 63 AND xUploadDone = FALSE THEN		// The transfer mode is active, but the values are not uploaded yet
				fbReadBitsFromWord(wData := awBusDataFromVTEM[0], iStartBit := 8, iEndBit := 12, iValue => iRecChannel);
				fbReadBitsFromWord(wData := awBusDataFromVTEM[0], iStartBit := 13, iEndBit := 15, iValue => iRecTransferCtrl);
				fbReadBitsFromWord(wData := awBusDataFromVTEM[1], iStartBit := 0, iEndBit := 7, iValue => iRecAddressedTargetType);
				fbReadBitsFromWord(wData := awBusDataFromVTEM[1], iStartBit := 8, iEndBit := 15, iValue => iRecIndex);
				iRecTransferValue := WORD_TO_INT(awBusDataFromVTEM[2]);
		 
				IF aTransferPackages[iCurrentValue].iChannel = iRecChannel AND iRecTransferCtrl = 2 AND aTransferPackages[iCurrentValue].iAddressedTarget = iRecAddressedTargetType AND
					aTransferPackages[iCurrentValue].iIndex = iRecIndex THEN
						// The addressed parameter was mirrored by the Motion Terminal, the uploaded value can be used
						aTransferPackages[iCurrentValue].iTransferValue := iRecTransferValue;
						
						xUploadError := FALSE;
						iCurrentValue := iCurrentValue +1;		// next value
						
						// check whether there is another value
						IF aTransferPackages[iCurrentValue].iAddressedTarget = 0 AND aTransferPackages[iCurrentValue].iChannel = 0 AND aTransferPackages[iCurrentValue].iIndex = 0 THEN 	// last value reached
										
							iCommandNumber := 2; 				// exit transfer mode
							iResponse := eTransferResponse.transfer_successful;
							xTransferComplete := TRUE;
							xStopPending := TRUE;
						ELSE
							iCommandNumber := 1; 				// command 'upload' for the (next) value
							iResponse := eTransferResponse.transferring;
						END_IF
				
				ELSIF iRecChannel = 0 AND iRecTransferCtrl = 0 AND iRecAddressedTargetType = 0 AND iRecIndex = 0 AND iRecTransferValue <> 0 AND xFirstCycle = FALSE THEN
					// An invalid command was sent when using the transfer mode
					// (Hint: At this point it cannot be identified if the invalid command was sent by this function block due to invalid inputs or if the
					// invalid command was created anywhere else. That's why the 'upload' command of the value in this function block is sent again.)
					
					xUploadError := TRUE;
					iCommandNumber := 1; 						// command 'upload' for the same value
					CASE iRecTransferValue OF	// indicates the type of the invalid command
						1: 	iResponse := eTransferResponse.invalid_Channel;
						2: 	iResponse := eTransferResponse.invalid_TransferControl;	// this should never happen 
						3: 	iResponse := eTransferResponse.invalid_AddressedTarget;
						4: 	iResponse := eTransferResponse.invalid_Index;
						5: 	iResponse := eTransferResponse.invalid_TransferValue;	// this cannot happen with an upload
						6: 	iResponse := eTransferResponse.invalid_combination;
						7:  iResponse := eTransferResponse.access_denied_DataInUse;
						8:	iResponse := eTransferResponse.no_data_empty_slot;
					END_CASE
					
				ELSE	// A different value is treated in transfer mode or the command was mirrored wrong
					// waiting for stop ack
					IF xStopPending = FALSE THEN
						iCommandNumber := 1; 			// command 'upload' for the current value
						iResponse := eTransferResponse.transferring;
						xUploadError := FALSE;
					END_IF
				END_IF
			
			ELSE // xUploadDone = TRUE
				IF aTransferPackages[iCurrentValue].iChannel = 0 AND aTransferPackages[iCurrentValue].iAddressedTarget = 0 AND  aTransferPackages[iCurrentValue].iIndex = 0 AND  aTransferPackages[iCurrentValue].iTransferValue = 0 THEN
					// The FB is still active although all values are already uploaded
					iResponse := eTransferResponse.transfer_successful;
					xUploadError := FALSE;
					iCommandNumber := 3; 			// do nothing (here: command 'stop', MAs remain stopped)
				ELSE
					// Another set of values was inserted to the FB without resetting the internal state with a falling edge at xExecute before
					iResponse := eTransferResponse.FB_needs_rising_edge_xExecute;
					xUploadError := TRUE;
					iCommandNumber := 2; 			// do nothing (here: command 'exit transfer mode')
				END_IF
			END_IF
		END_IF
	
	ELSE // xInputValid = FALSE OR xInputConsistent = FALSE
		xUploadDone := FALSE;
		xUploadError := TRUE;
		IF iRecValveMode = 63 THEN
			iCommandNumber := 2; 				// command 'exit transfer mode'
		ELSE
			iCommandNumber := 3;				// command 'stop'
		END_IF
	END_IF
		
	xFirstCycle := FALSE;

ELSIF xExecute = FALSE AND xFirstCycle = FALSE THEN	// falling edge at input xExecute, reseting the function block
	IF iRecValveMode = 63 THEN
		iCommandNumber := 2;						// exit transfer mode
	ELSE
		xFirstCycle := TRUE;
		xUploadDone := FALSE;
		xUploadError := FALSE;
		xTransferComplete := FALSE;
		iCurrentValue := 0;
		xStopPending := FALSE;
		iResponse := eTransferResponse.ready_for_new_transfer;
		iCommandNumber := 0;						// do nothing (idle)		
	END_IF

ELSIF xExecute = FALSE AND xFirstCycle = TRUE THEN	// idle mode for the function block
	iResponse := eTransferResponse.ready_for_new_transfer;
	iCommandNumber := 0;
END_IF

CASE iCommandNumber OF
	0: // idle

	1: // upload the current value, addressed and specified in the array of values
		fbWriteValueToWord(iValue := 63, iStartBit := 0, iEndBit := 5, wDataWord := awBusDataToVTEM[0]); 												// ValveMode = 63
		fbWriteValueToWord(iValue := 0, iStartBit := 6, iEndBit := 7, wDataWord := awBusDataToVTEM[0]); 												// (empty)
		fbWriteValueToWord(iValue := aTransferPackages[iCurrentValue].iChannel, iStartBit := 8, iEndBit := 12, wDataWord := awBusDataToVTEM[0]); 		// Channel
		fbWriteValueToWord(iValue := 2, iStartBit := 13, iEndBit := 15, wDataWord := awBusDataToVTEM[0]); 												// TransferControl = upload
		fbWriteValueToWord(iValue := aTransferPackages[iCurrentValue].iAddressedTarget, iStartBit := 0, iEndBit := 7, wDataWord := awBusDataToVTEM[1]); // AddressedTarget
		fbWriteValueToWord(iValue := aTransferPackages[iCurrentValue].iIndex, iStartBit := 8, iEndBit := 15, wDataWord := awBusDataToVTEM[1]); 			// Index
		
		awBusDataToVTEM[2] := 0;
	
	2: // exit transfer mode
		fbWriteValueToWord(iValue := 63, iStartBit := 0, iEndBit := 5, wDataWord := awBusDataToVTEM[0]); 												// ValveMode = 63
		fbWriteValueToWord(iValue := 0, iStartBit := 6, iEndBit := 7, wDataWord := awBusDataToVTEM[0]); 												// (empty)
		fbWriteValueToWord(iValue := 0, iStartBit := 8, iEndBit := 12, wDataWord := awBusDataToVTEM[0]); 												// Channel
		fbWriteValueToWord(iValue := 3, iStartBit := 13, iEndBit := 15, wDataWord := awBusDataToVTEM[0]); 												// TransferControl = exit

		awBusDataToVTEM[1] := 0;
		awBusDataToVTEM[2] := 0;

	3: // stop all Motion Apps
		fbWriteValueToWord(iValue := 61, iStartBit := 0, iEndBit := 5, wDataWord := awBusDataToVTEM[0]); 												// ValveMode = 61
		fbWriteValueToWord(iValue := 0, iStartBit := 6, iEndBit := 15, wDataWord := awBusDataToVTEM[0]); 												// (empty)

		awBusDataToVTEM[1] := 0;
		awBusDataToVTEM[2] := 0;
END_CASE

END_FUNCTION_BLOCK

// Transfermode/FB_Upload_Single_Parameter
/// This function block can be used to run the transfer mode of the Motion Terminal in order to upload a single value.
/// The value to be uploaded needs to be addressed, indicating the channel, the addressed target and the index of the value.

FUNCTION_BLOCK FB_Upload_Single_Parameter
VAR_INPUT
	awBusDataFromVTEM 		: ARRAY [0..2] OF WORD; 		(* 6 bytes of process data received from the Motion Terminal *)
END_VAR

VAR_IN_OUT
	awBusDataToVTEM			: ARRAY [0..2] OF WORD; 		(* 6 bytes of process data sent to the Motion Terminal *)
END_VAR

VAR_INPUT	
	xExecute 				: BOOL;							(* has to be set to TRUE for an upload and to FALSE to reset the function block after an upload *)
	
	iChannel 				: INT;							(* the channel the value is to be read from (see documentation for details) *)
	iAddressedTarget 		: INT; 							(* the target by which the parameter is used (was "iAddressedApp" in former versions) (see documentation for details) *)
	iIndex 					: INT;							(* the index of the parameter (see documentation for details) *)
END_VAR

VAR_OUTPUT
	iResponse 				: eTransferResponse;			(* returns the status of the execution of the upload process *)
	iUploadedValue 			: INT := 0;  					(* the uploaded value *)
	
	xUploadDone 			: BOOL; 						(* indicates whether the upload was successful *)
	xUploadError 			: BOOL; 						(* indicates whether an error occurred during the transfer *)
END_VAR

VAR
	iRecValveMode 			: INT;
	iRecValveStatus 		: eValveState;
	iCommandNumber			: INT; 							(* indicates the command to be executed *)

	fbWriteValueToWord		: FB_Write_Value_To_Word;
	fbReadBitsFromWord 		: FB_Read_Bits_From_Word;
	iRecChannel				: INT;
	iRecTransferCtrl		: INT;
	iRecAddressedTarget		: INT;
	iRecIndex				: INT;
	iRecUploadedValue		: INT;
	
	iAppStatus				: INT;
	iLastIndex				: INT;
	iLastChannel			: INT;
	iLastAddressedTarget	: INT;
	xFirstCycle				: BOOL := TRUE;
	xTransferComplete		: BOOL;
	iFCChannel				: INT;
	iFCAddressedTarget		: INT;
	iFCIndex				: INT;
	xInputValid				: BOOL;
	xInputConsistent		: BOOL;
END_VAR

(*****************************************************************************************************

Festo SE & Co. KG, Esslingen
Copyright (c) 2018. All rights reserved.

Product:            Motion Terminal VTEM
Description:        Function block to upload a single parameter from the Motion Terminal

